			SP_RunStp50: // Do cleaning and reload from lift
				eRestartStep := SP_RunStp50;
				eRestartLoaderStep := SP_RunStp50;
				IF sRunData.sStatusLoader = RS_WaitRequest THEN
					// Check if table can be cleaned
					IF sRunData.sStatusTable = RS_WaitRequest AND NOT bTableIsClean THEN
						// Clean the table
						sRunData.eCmdTable := RCT_Clean;
					END_IF
					IF bNeedNewPart THEN			// HFO : add "or sProdLot.dProdQty < sProdLot.dLotQty" to pearl the 2 last pieces
						IF NOT sRunData.TDataLoader.aTPartData[0].bPartPresent AND NOT bTablePos2NeedPart THEN
							sRunData.TDataLoader.eModule := LMP_Lift1;
							sRunData.TDataLoader.eTaker := LH_Head1;
							sRunData.eCmdLoader := RCLo_PrepareTakePart;
							eManagerStep := SP_RunStp55;
						ELSIF NOT sRunData.TDataLoader.aTPartData[1].bPartPresent THEN
							sRunData.TDataLoader.eModule := LMP_Lift1;
							sRunData.TDataLoader.eTaker := LH_Head2;
							sRunData.eCmdLoader := RCLo_PrepareTakePart;
							eManagerStep := SP_RunStp55;
						ELSIF sRunData.sStatusTable = RS_WaitRequest THEN
							bTableIsClean := TRUE;
							eManagerStep := SP_RunStp70;
						END_IF	
					ELSIF sRunData.sStatusTable = RS_WaitRequest AND sProdLot.dProdQty < sProdLot.dLotQty THEN			// TODO : HFO, add elseif to pearl the 2 last pieces
						bTableIsClean := TRUE;
						eManagerStep := SP_RunStp70;
					ELSE
						eManagerStep := SP_RunStp80;
						// eManagerStep := SP_RunStp160; 	// purging
					END_IF
				END_IF				
			SP_RunStp55:
				IF sRunData.sStatusLoader = RS_WaitRequest THEN
					sRunData.eCmdLoader := RCLo_TakePart;
					eManagerStep := SP_RunStp60;
				END_IF
			SP_RunStp60:
				IF sRunData.sStatusLoader = RS_WaitRequest 
						AND sRunData.sStatusTable = RS_WaitRequest THEN
					bTableIsClean := TRUE;
					eManagerStep := SP_RunStp50;
				END_IF
			SP_RunStp70: (* Drop part on layering *)
				IF sRunData.sStatusTable = RS_WaitRequest THEN
					eRestartStep := SP_RunStp70;
					eRestartLoaderStep := SP_RunStp70;
					IF sRunData.TDataLoader.aTPartData[0].bPartPresent THEN
						IF sRunData.TDataLoader.aTPartData[0].bToReject THEN
							sRunData.TDataLoader.eModule := LMP_Reject;
							sRunData.TDataLoader.eTaker := LH_Head1;
							sRunData.eCmdLoader := RCLo_PrepareDropPart;
							eManagerStep := SP_RunStp150;
						ELSE
							sRunData.TDataLoader.eModule := LMP_Table;
							sRunData.TDataLoader.eTaker := LH_Head1;
							sRunData.TDataLoader.iLayringPos := 0;
							sRunData.eCmdLoader := RCLo_PrepareDropPart;
							eManagerStep := SP_RunStp75;
						END_IF
					ELSIF sRunData.TDataLoader.aTPartData[1].bPartPresent THEN
						IF sRunData.TDataLoader.aTPartData[1].bToReject THEN
							sRunData.TDataLoader.eModule := LMP_Reject;
							sRunData.TDataLoader.eTaker := LH_Head2;
							sRunData.eCmdLoader := RCLo_PrepareDropPart;
							bTablePos2NeedPart := TRUE;
							eManagerStep := SP_RunStp150;
						ELSE
							sRunData.TDataLoader.eModule := LMP_Table;
							sRunData.TDataLoader.eTaker := LH_Head2;
							sRunData.TDataLoader.iLayringPos := 1;
							sRunData.eCmdLoader := RCLo_PrepareDropPart;
							bTablePos2NeedPart := FALSE;
							eManagerStep := SP_RunStp75;
						END_IF
					ELSE
						// Loading finished, turn table
						eManagerStep := SP_RunStp80;
					END_IF
				END_IF
			SP_RunStp75:
				IF sRunData.sStatusLoader = RS_WaitRequest THEN
					sRunData.TDataTable.iGiveTakeLayeringPosition := sRunData.TDataLoader.iLayringPos;
					sRunData.eCmdLoader := RCLo_GivePart;
					sRunData.eCmdTable := RCT_TakePart;
					eManagerStep := SP_RunStp77;
				END_IF
			SP_RunStp77:
				IF sRunData.sStatusLoader = RS_WaitRequest AND  sRunData.sStatusTable = RS_WaitRequest  THEN
					eManagerStep := SP_RunStp70;
				END_IF		
			SP_RunStp80:
				IF sRunData.sStatusLoader = RS_WaitRequest AND  sRunData.sStatusTable = RS_WaitRequest  THEN
					sRunData.eCmdLoader := RCLo_MoveToSafe;
					eManagerStep := SP_RunStp85;
				END_IF		
			SP_RunStp85:
				IF sRunData.sStatusLoader = RS_WaitRequest AND bPearlingFinishOnTableSide THEN
					(* Pearling finish *)
					bReadyForPearling := FALSE;
					eManagerStep := SP_RunStp90;
				END_IF
			SP_RunStp90:
				eRestartStep := SP_RunStp96;
				eRestartLoaderStep := SP_RunStp93;
				sRunData.eCmdTable := RCT_Turn;
				eWorkingTableSide := ePearlingTableSide;
				eManagerStep := SP_RunStp93;
			SP_RunStp93: (*Turning Table *)
				IF sRunData.sStatusTable = RS_ProcessRequest2 THEN
					IF iPartOnProcess = 0 AND NOT bNeedNewPart THEN
						eManagerStep := SP_RunStp300;
					ELSE
						bReadyForPearling := TRUE;
						eManagerStep := SP_RunStp96;
					END_IF
				END_IF
			SP_RunStp96: (*Cleaning Table *)
				IF sRunData.sStatusTable = RS_WaitRequest  AND  sRunData.sStatusLoader = RS_WaitRequest  THEN
					bTableIsClean := TRUE;
					eManagerStep := SP_RunStp1;
				END_IF
			SP_RunStp100: (* Unloading part on layering *)
				IF sRunData.TDataTable.aTPartData[0,0,sRunData.TDataTable.eTableSide].bPartPresent OR sRunData.TDataTable.aTPartData[1,0,sRunData.TDataTable.eTableSide].bPartPresent THEN
					eRestartStep := SP_RunStp100;
					eRestartLoaderStep := SP_RunStp100;
					sRunData.TDataLoader.eModule := LMP_Table;
					sRunData.eCmdLoader := RCLo_PrepareTakePart;
					eManagerStep := SP_RunStp105;
				ELSE
					eManagerStep := SP_RunStp1;
				END_IF
			SP_RunStp105:
				IF sRunData.sStatusLoader = RS_WaitRequest THEN
					sRunData.eCmdLoader := RCLo_TakePart;
					sRunData.TDataTable.iGiveTakeLayeringPosition := sRunData.TDataLoader.iLayringPos;
					sRunData.TDataTable.iGiveTakeLayeringOffsetPosition := sRunData.TDataLoader.iLayringOffsetPos;
					sRunData.eCmdTable := RCT_GivePart;
					eManagerStep := SP_RunStp110;
				END_IF
			SP_RunStp110:
				IF sRunData.sStatusLoader = RS_WaitRequest AND  sRunData.sStatusTable = RS_WaitRequest  THEN
					eManagerStep := SP_RunStp1;
				END_IF
			SP_RunStp150: // Give bad part to the reject
				IF sRunData.sStatusLoader = RS_WaitRequest THEN
					sRunData.eCmdLoader := RCLo_GivePart;
					eManagerStep := SP_RunStp151;
				END_IF
			SP_RunStp151:
				IF sRunData.sStatusLoader = RS_WaitRequest THEN
					eManagerStep := SP_RunStp50;
				END_IF
			SP_RunStp160: // TODO : (HFO) // Steps for purging 
				IF sRunData.sStatusLoader = RS_WaitRequest AND  sRunData.sStatusTable = RS_WaitRequest  THEN
					sRunData.eCmdLoader := RCLo_MoveToSafe;
					//eManagerStep := SP_RunStp85;
				END_IF		
			SP_RunStp200:
				IF sRunData.sStatusLoader = RS_WaitRequest THEN
					IF sRunData.TDataLoader.aTPartData[LH_Head1].bToReject THEN
						sRunData.TDataLoader.eModule := LMP_Reject;
					ELSIF sProductionCmd.TRequestSample.Activate THEN
						sRunData.TDataLoader.eModule := LMP_Sample;
						sProductionCmd.TRequestSample.Activate := FALSE;
					ELSE
						sProductionCmd.TAutoSampling.iPeriodCnt := sProductionCmd.TAutoSampling.iPeriodCnt + 1;
						IF sProductionCmd.TAutoSampling.bEnable AND (sProductionCmd.TAutoSampling.iPeriodCnt >= (sProductionCmd.TAutoSampling.iPeriod - sProductionCmd.TAutoSampling.iBatchSize)) THEN
							sRunData.TDataLoader.eModule := LMP_Sample;
							sProductionCmd.TAutoSampling.iBatchCnt := sProductionCmd.TAutoSampling.iBatchCnt + 1;
							IF sProductionCmd.TAutoSampling.iBatchCnt >= sProductionCmd.TAutoSampling.iBatchSize THEN
								sProductionCmd.TAutoSampling.iBatchCnt := 0;
								sProductionCmd.TAutoSampling.iPeriodCnt := 0;
							END_IF
						ELSE
							sRunData.TDataLoader.eModule := LMP_Lift2;
						END_IF
					END_IF
					sRunData.eCmdLoader := RCLo_PrepareDropPart;
					eManagerStep := SP_RunStp205;
				END_IF
			SP_RunStp205:
				IF sRunData.sStatusLoader = RS_WaitRequest THEN
					sRunData.eCmdLoader := RCLo_GivePart;
					eManagerStep := SP_RunStp210;
				END_IF
			SP_RunStp210:
				IF sRunData.sStatusLoader = RS_WaitRequest THEN
					bTableIsClean := TRUE;
					eManagerStep := SP_RunStp2;
				END_IF
			SP_RunStp300: (*End of recipe *)
				bReadyForPearling := FALSE;
				sRunData.eCmdLoader := RCLo_EndOfRecipe;
				eManagerStep := SP_RunStp305;
			SP_RunStp305: (*Loader in safe and lift in unload position *)
				IF sRunData.sStatusLoader = RS_WaitRequest  AND sRunData.sStatusPearling = RS_WaitRequest AND sRunData.sStatusTable = RS_WaitRequest THEN
					eManagerStep := SP_RunStp0;
				END_IF
		END_CASE
	ELSE
		CASE eManagerStep OF
			SP_InitStp1:	(*Recovery, Drop plate if we have one*)
				sRunData.eCmdPearling := RCP_CheckSharpen;
				bReadyForPearling := FALSE;
				bTableIsClean := FALSE;
				IF sRunData.TDataLoader.bPlatePresent THEN
					sRunData.eCmdLoader := RCLo_SwitchPlate;
					eManagerStep := SP_InitStp2;
				ELSE
					eManagerStep := SP_InitStp3;
				END_IF
			SP_InitStp2: (* Switch plate done *)
				IF sRunData.sStatusLoader = RS_WaitRequest THEN
					eManagerStep := SP_InitStp3;
				END_IF
			SP_InitStp3: (* Do we need a table turn ? *)
				IF  sRunData.TDataTable.eTableSide <>  eWorkingTableSide THEN
					sRunData.eCmdTable := RCT_Turn;
					eManagerStep := SP_InitStp4;
				ELSE
					eManagerStep := SP_InitStp5;
				END_IF
			SP_InitStp4:
					IF sRunData.sStatusTable = RS_WaitRequest THEN
						eManagerStep := SP_InitStp5;
					END_IF
			SP_InitStp5:
				bReadyForPearling := TRUE;
				IF sRunData.TDataLoader.aTPartData[LH_Head1].bPartPresent THEN
					eManagerStep := eRestartLoaderStep;
				ELSE
					eManagerStep := eRestartStep;
				END_IF
	(* Running Step *)
			SP_RunStp1:
				eRestartStep := SP_RunStp1;
				eRestartLoaderStep := SP_RunStp7;
				iRunLayering := 0;
				iRunLayeringOffset := 0;
				bLastPart := FALSE;
				eManagerStep := SP_RunStp3;
			SP_RunStp2:
				bLastPart := FALSE;
				IF bLayeringWithTwoParts THEN
					IF iRunLayering=0 AND iRunLayeringOffset=0 THEN
						iRunLayering := 0;
						iRunLayeringOffset := 1;
						eManagerStep := SP_RunStp3;
					ELSIF iRunLayering=0 AND iRunLayeringOffset=1 THEN
						iRunLayering := 1;
						iRunLayeringOffset := 0;
						eManagerStep := SP_RunStp3;
					ELSIF iRunLayering=1 AND iRunLayeringOffset=0 THEN
						iRunLayering := 1;
						iRunLayeringOffset := 1;
						bLastPart := TRUE;
						eManagerStep := SP_RunStp3;
					ELSE
						eManagerStep := SP_RunStp20;
					END_IF
				ELSE
					IF iRunLayering=0 AND iRunLayeringOffset=0 THEN
						iRunLayering := 1;
						iRunLayeringOffset := 0;
						bLastPart := TRUE;
						eManagerStep := SP_RunStp3;
					ELSE
						eManagerStep := SP_RunStp20;
					END_IF
				END_IF
			SP_RunStp3:
				IF sRunData.TDataTable.aTPartData[iRunLayering,iRunLayeringOffset,sRunData.TDataTable.eTableSide].bPartPresent THEN
					bTableIsClean := FALSE;
					eManagerStep := SP_RunStp4;
				ELSE
					eManagerStep := SP_RunStp2; (* Skip *)
				END_IF
			SP_RunStp4: (* Unloading part on layering*)
				sRunData.TDataLoader.eModule := LMP_Table;
				sRunData.TDataLoader.eTaker := LH_Head1;
				sRunData.TDataLoader.iLayringPos := iRunLayering;
				sRunData.TDataLoader.iLayringOffsetPos := iRunLayeringOffset;
				sRunData.eCmdLoader := RCLo_PrepareTakePart;
				eManagerStep := SP_RunStp5;
			SP_RunStp5:
				IF sRunData.sStatusLoader = RS_WaitRequest THEN
					sRunData.eCmdLoader := RCLo_TakePart;
					sRunData.TDataTable.iGiveTakeLayeringPosition := sRunData.TDataLoader.iLayringPos;
					sRunData.TDataTable.iGiveTakeLayeringOffsetPosition := sRunData.TDataLoader.iLayringOffsetPos;
					sRunData.eCmdTable := RCT_GivePart;
					eManagerStep := SP_RunStp6;
				END_IF
			SP_RunStp6:
				IF sRunData.sStatusLoader = RS_WaitRequest AND  sRunData.sStatusTable = RS_WaitRequest  THEN
					IF bLastPart AND NOT bTableIsClean THEN
						sRunData.eCmdLoader := RCLo_MoveToSafe;
					END_IF
					eManagerStep := SP_RunStp7;
				END_IF
			SP_RunStp7:
				IF sRunData.sStatusLoader = RS_WaitRequest THEN
					IF bLastPart AND NOT bTableIsClean THEN
						sRunData.eCmdTable := RCT_Clean;
					END_IF
					IF sRunData.TDataLoader.aTPartData[LH_Head1].bToReject THEN
						sRunData.TDataLoader.eModule := LMP_Reject;
					ELSIF sProductionCmd.TRequestSample.Activate THEN
						sRunData.TDataLoader.eModule := LMP_Sample;
						sProductionCmd.TRequestSample.Activate := FALSE;
					ELSE
						sProductionCmd.TAutoSampling.iPeriodCnt := sProductionCmd.TAutoSampling.iPeriodCnt + 1;
						IF sProductionCmd.TAutoSampling.bEnable AND (sProductionCmd.TAutoSampling.iPeriodCnt >= (sProductionCmd.TAutoSampling.iPeriod - sProductionCmd.TAutoSampling.iBatchSize)) THEN
							sRunData.TDataLoader.eModule := LMP_Sample;
							sProductionCmd.TAutoSampling.iBatchCnt := sProductionCmd.TAutoSampling.iBatchCnt + 1;
							IF sProductionCmd.TAutoSampling.iBatchCnt >= sProductionCmd.TAutoSampling.iBatchSize THEN
								sProductionCmd.TAutoSampling.iBatchCnt := 0;
								sProductionCmd.TAutoSampling.iPeriodCnt := 0;
							END_IF
						ELSE
							sRunData.TDataLoader.eModule := LMP_Lift2;
						END_IF
					END_IF
					sRunData.eCmdLoader := RCLo_PrepareDropPart;
					eManagerStep := SP_RunStp9;
				END_IF
			SP_RunStp9:
				IF sRunData.sStatusLoader = RS_WaitRequest THEN
					sRunData.eCmdLoader := RCLo_GivePart;
					eManagerStep := SP_RunStp10;
				END_IF
			SP_RunStp10:
				IF sRunData.sStatusLoader = RS_WaitRequest THEN
					IF bUse103171OptimA1  THEN
						eManagerStep := SP_RunStp11;
					ELSE
						IF sRunData.sStatusTable = RS_WaitRequest THEN
							bTableIsClean := TRUE;
							eManagerStep := SP_RunStp2;
						END_IF
					END_IF
				END_IF
			SP_RunStp11: (* During cleaning, load part on head 2*)
				eRestartStep := SP_RunStp11;
				eRestartLoaderStep := SP_RunStp11;
				IF iPartOnProcess = 0 AND NOT bNeedNewPart THEN
					eManagerStep := SP_RunStp100;
				ELSE
					eManagerStep := SP_RunStp12;
				END_IF
			SP_RunStp12:
				sRunData.TDataLoader.eModule := LMP_Lift1;
				sRunData.TDataLoader.eTaker := LH_Head1;
				sRunData.eCmdLoader := RCLo_PrepareTakePart;
				eManagerStep := SP_RunStp13;
			SP_RunStp13:
				IF sRunData.sStatusLoader = RS_WaitRequest THEN
					sRunData.eCmdLoader := RCLo_TakePart;
					eManagerStep := SP_RunStp14;
				END_IF
			SP_RunStp14:
				IF sRunData.sStatusLoader = RS_WaitRequest THEN
					(* Check if table has finished or not *)
					IF sRunData.sStatusTable = RS_WaitRequest THEN
						eManagerStep := SP_RunStp2;
					ELSIF bUse103171OptimB5PreMoveXY THEN
						(* Move to safe to save time *)
						eManagerStep := SP_RunStp15;
					END_IF
				END_IF
			SP_RunStp15:
				eRestartStep := SP_RunStp15;
				eRestartLoaderStep := SP_RunStp15;
				sRunData.eCmdLoader := RCLo_MoveToSafe;
				eManagerStep := SP_RunStp16;
			SP_RunStp16:
				IF sRunData.sStatusLoader = RS_WaitRequest AND sRunData.sStatusTable = RS_WaitRequest THEN
					eManagerStep := SP_RunStp2;
				END_IF
	
			SP_RunStp20: (* Unloading finish, proceed cleaning*)
				eRestartStep := SP_RunStp20;
				eRestartLoaderStep := SP_RunStp20;
				IF iPartOnProcess = 0 AND NOT bNeedNewPart THEN
					eManagerStep := SP_RunStp100;
				ELSIF sRunData.sStatusTable = RS_WaitRequest THEN
					sRunData.eCmdLoader := RCLo_MoveToSafe;
					eManagerStep := SP_RunStp21;
				ELSE
					eManagerStep := SP_RunStp21;
				END_IF
			SP_RunStp21:
				IF sRunData.sStatusLoader = RS_WaitRequest THEN
					IF NOT bTableIsClean THEN
						sRunData.eCmdTable := RCT_Clean;
					END_IF
					IF bUse103171OptimA1 AND NOT sRunData.TDataLoader.aTPartData[LH_Head2].bPartPresent THEN
						eManagerStep := SP_RunStp200;
					ELSE
						eManagerStep := SP_RunStp22;
					END_IF
				END_IF
			SP_RunStp22: (*Cleaning Table*)
				IF sRunData.sStatusTable = RS_WaitRequest THEN
					bTableIsClean := TRUE;
					eManagerStep := SP_RunStp40;
				END_IF
			SP_RunStp40: (* Load layering *)
				eRestartStep := SP_RunStp40;
				eRestartLoaderStep := SP_RunStp44;
				iRunLayering := -1;
				iRunLayeringOffset := 1;
				eManagerStep := SP_RunStp41;
			SP_RunStp41:
				IF bLayeringWithTwoParts THEN
					IF bNeedNewPart OR iRunLayeringOffset=0 THEN
						IF iRunLayering=-1 THEN
							iRunLayering := 0;
							iRunLayeringOffset := 0;
							eManagerStep := SP_RunStp42;
						ELSIF iRunLayering=0 AND iRunLayeringOffset=0 THEN
							iRunLayering := 0;
							iRunLayeringOffset := 1;
							eManagerStep := SP_RunStp42;
						ELSIF iRunLayering=0 AND iRunLayeringOffset=1 THEN
							iRunLayering := 1;
							iRunLayeringOffset := 0;
							eManagerStep := SP_RunStp42;
						ELSIF iRunLayering=1 AND iRunLayeringOffset=0 THEN
							iRunLayering := 1;
							iRunLayeringOffset := 1;
							eManagerStep := SP_RunStp42;
						ELSE
							eManagerStep := SP_RunStp50;
						END_IF
					ELSE
						eManagerStep := SP_RunStp50;
					END_IF
				ELSE
					IF bNeedNewPart THEN
						IF iRunLayering=-1 THEN
							iRunLayering := 0;
							iRunLayeringOffset := 0;
							eManagerStep := SP_RunStp42;
						ELSIF iRunLayering=0 AND iRunLayeringOffset=0 THEN
							iRunLayering := 1;
							iRunLayeringOffset := 0;
							eManagerStep := SP_RunStp42;
						ELSE
							eManagerStep := SP_RunStp50;
						END_IF
					ELSE
						eManagerStep := SP_RunStp50;
					END_IF
				END_IF
			SP_RunStp42:
				IF NOT sRunData.TDataTable.aTPartData[iRunLayering,iRunLayeringOffset,sRunData.TDataTable.eTableSide].bPartPresent THEN
					bTableIsClean := FALSE;
					sRunData.TDataLoader.eModule := LMP_Lift1;
					sRunData.TDataLoader.eTaker := LH_Head1;
					sRunData.eCmdLoader := RCLo_PrepareTakePart;
					eManagerStep := SP_RunStp43;
				ELSE
					eManagerStep := SP_RunStp41; (* Skip *)
				END_IF
			SP_RunStp43:
				IF sRunData.sStatusLoader = RS_WaitRequest THEN
					sRunData.eCmdLoader := RCLo_TakePart;
					eManagerStep := SP_RunStp44;
				END_IF
			SP_RunStp44:
				IF sRunData.sStatusLoader = RS_WaitRequest THEN
					(* Check if a part was taken or not *)
					IF sRunData.TDataLoader.aTPartData[LH_Head1].bPartPresent THEN
						sRunData.TDataLoader.eModule := LMP_Table;
						sRunData.TDataLoader.iLayringPos := iRunLayering;
						sRunData.TDataLoader.iLayringOffsetPos := iRunLayeringOffset;
						sRunData.eCmdLoader := RCLo_PrepareDropPart;
						eManagerStep := SP_RunStp45;
					ELSE
						eManagerStep := SP_RunStp42;
					END_IF
				END_IF
			SP_RunStp45:
				IF sRunData.sStatusLoader = RS_WaitRequest THEN
					sRunData.eCmdLoader := RCLo_GivePart;
					sRunData.TDataTable.iGiveTakeLayeringPosition := sRunData.TDataLoader.iLayringPos;
					sRunData.TDataTable.iGiveTakeLayeringOffsetPosition := sRunData.TDataLoader.iLayringOffsetPos;
					sRunData.eCmdTable := RCT_TakePart;
					eManagerStep := SP_RunStp46;
				END_IF
			SP_RunStp46:
				IF sRunData.sStatusLoader = RS_WaitRequest AND  sRunData.sStatusTable = RS_WaitRequest  THEN
					(* Reject part if not correctly dropped *)
					IF sRunData.TDataLoader.aTPartData[LH_Head2].bPartPresent THEN
						eManagerStep := SP_RunStp47;
					ELSE
						eManagerStep := SP_RunStp41;
					END_IF
				END_IF
			SP_RunStp47:
				sRunData.TDataLoader.eModule := LMP_Reject;
				sRunData.eCmdLoader := RCLo_PrepareDropPart;
				eManagerStep := SP_RunStp48;
			SP_RunStp48:
				IF sRunData.sStatusLoader = RS_WaitRequest THEN
					sRunData.eCmdLoader := RCLo_GivePart;
					eManagerStep := SP_RunStp49;
				END_IF
			SP_RunStp49:
				IF sRunData.sStatusLoader = RS_WaitRequest THEN
					eManagerStep := SP_RunStp42;
				END_IF
			SP_RunStp50: (* Launch loader to safe *)
				eRestartStep := SP_RunStp50;
				eRestartLoaderStep := SP_RunStp50;
				sRunData.eCmdLoader := RCLo_MoveToSafe;
				eManagerStep := SP_RunStp51;
			SP_RunStp51:
				IF sRunData.sStatusLoader = RS_WaitRequest AND bPearlingFinishOnTableSide THEN
					(* Pearling finish *)
					bReadyForPearling := FALSE;
					eManagerStep := SP_RunStp52;
				END_IF
			SP_RunStp52:
				eRestartStep := SP_RunStp54;
				eRestartLoaderStep := SP_RunStp53;
				IF bDisableCleanAfterPearling  THEN
					sRunData.eCmdTable := RCT_Turn;
				ELSE
					sRunData.eCmdTable := RCT_TurnAndClean;
				END_IF
				eWorkingTableSide := ePearlingTableSide;
				eManagerStep := SP_RunStp53;
			SP_RunStp53: (*Turning Table *)
				IF sRunData.sStatusTable = RS_ProcessRequest2 THEN
					bReadyForPearling := TRUE;
					eManagerStep := SP_RunStp54;
				END_IF
			SP_RunStp54: (*Cleaning Table *)
				IF sRunData.sStatusTable = RS_WaitRequest  AND  sRunData.sStatusLoader = RS_WaitRequest  THEN
					bTableIsClean := TRUE;
					eManagerStep := SP_RunStp1;
				END_IF
			SP_RunStp100: (*End of recipe *)
				bReadyForPearling := FALSE;
				sRunData.eCmdLoader := RCLo_EndOfRecipe;
				eManagerStep := SP_RunStp101;
			SP_RunStp101: (*Loader in safe and lift in unload position *)
				IF sRunData.sStatusLoader = RS_WaitRequest  AND sRunData.sStatusPearling = RS_WaitRequest AND sRunData.sStatusTable = RS_WaitRequest THEN
					eManagerStep := SP_RunStp0;
				END_IF
	
			SP_RunStp200: (* During cleaning, load part on head 2*)
				eRestartStep := SP_RunStp200;
				eRestartLoaderStep := SP_RunStp200;
				IF iPartOnProcess = 0 AND NOT bNeedNewPart THEN
					eManagerStep := SP_RunStp100;
				ELSE
					eManagerStep := SP_RunStp240;
				END_IF
			SP_RunStp240: (* Load part on head 2 to save time*)
				eRestartStep := SP_RunStp240;
				eRestartLoaderStep := SP_RunStp244;
				eManagerStep := SP_RunStp241;
			SP_RunStp241:
				sRunData.TDataLoader.eModule := LMP_Lift1;
				sRunData.TDataLoader.eTaker := LH_Head2;
				sRunData.eCmdLoader := RCLo_PrepareTakePart;
				eManagerStep := SP_RunStp242;
			SP_RunStp242:
				IF sRunData.sStatusLoader = RS_WaitRequest THEN
					sRunData.eCmdLoader := RCLo_TakePart;
					eManagerStep := SP_RunStp244;
				END_IF
			SP_RunStp244:
				IF sRunData.sStatusLoader = RS_WaitRequest THEN
					(* Check if table has finished or not *)
					IF sRunData.sStatusTable = RS_WaitRequest THEN
						eManagerStep := SP_RunStp1;
					ELSIF bUse103171OptimB5PreMoveXY THEN
						(* Move to safe to save time *)
						eManagerStep := SP_RunStp245;
					END_IF
				END_IF
			SP_RunStp245:
				eRestartStep := SP_RunStp245;
				eRestartLoaderStep := SP_RunStp245;
				sRunData.eCmdLoader := RCLo_MoveToSafe;
				eManagerStep := SP_RunStp246;
			SP_RunStp246:
				IF sRunData.sStatusLoader = RS_WaitRequest AND sRunData.sStatusTable = RS_WaitRequest THEN
					eManagerStep := SP_RunStp1;
				END_IF
		END_CASE
	END_IF
	IF bLayeringWithTwoParts THEN
		IF bSimPearling AND  bReadyForPearling THEN
			IF sRunData.TDataTable.aTPartData[0,0,ePearlingTableSide].bPartPresent THEN
				sRunData.TDataTable.aTPartData[0,0,ePearlingTableSide].abPearlingDone[0,PS_SUS] := TRUE;
			END_IF
			IF sRunData.TDataTable.aTPartData[0,1,ePearlingTableSide].bPartPresent THEN
				sRunData.TDataTable.aTPartData[0,1,ePearlingTableSide].abPearlingDone[0,PS_SUS] := TRUE;
			END_IF
			IF sRunData.TDataTable.aTPartData[1,0,ePearlingTableSide].bPartPresent THEN
				sRunData.TDataTable.aTPartData[1,0,ePearlingTableSide].abPearlingDone[0,PS_SUS] := TRUE;
			END_IF
			IF sRunData.TDataTable.aTPartData[1,1,ePearlingTableSide].bPartPresent THEN
				sRunData.TDataTable.aTPartData[1,1,ePearlingTableSide].abPearlingDone[0,PS_SUS] := TRUE;
			END_IF
		ELSIF  NOT bSimPearling AND sRunData.sStatusPearling = RS_WaitRequest  AND  bReadyForPearling THEN
			IF sConfigFileData.bParallelProduction THEN
				(* Pearling does nothing, launch pearling if there is part to pearl *)
				sRunData.TDataPearling.abUseSpindle[PH_Left] := FALSE;
				sRunData.TDataPearling.abUseSpindle[PH_Right] := FALSE;
				sRunData.TDataPearling.bForceSharpenAfterPearling := FALSE;
				FOR iLayeringOffsetPos := 0 TO iMaxLayeringOffsetPos DO
					sRunData.TDataPearling.sPearlingData := sConfigFileData.asPearlingData[PS_SUS].THead[PH_Left]; (* Always same recipe when parrelle prod *)
					IF sRunData.TDataTable.aTPartData[0,iLayeringOffsetPos,ePearlingTableSide].bPartPresent AND
						sRunData.TDataPearling.abUseSpindle[PH_Left] = FALSE AND sRunData.TDataPearling.abUseSpindle[PH_Right] = FALSE AND
						NOT (sRunData.TDataTable.aTPartData[0,iLayeringOffsetPos,ePearlingTableSide].abPearlingDone[0,PS_SUS] OR sRunData.TDataTable.aTPartData[0,iLayeringOffsetPos,ePearlingTableSide].abPearlingDone[1,PS_SUS]) THEN
						sRunData.TDataPearling.abUseSpindle[PH_Left] := TRUE;
						sRunData.TDataPearling.iLayringPos := 0;
						sRunData.TDataPearling.iLayringOffsetPos := iLayeringOffsetPos;
						sRunData.TDataPearling.apsPartData[PH_Left] := ADR(sRunData.TDataTable.aTPartData[0,iLayeringOffsetPos,ePearlingTableSide]);
						IF sRunData.TDataTable.aTPartData[1,iLayeringOffsetPos,ePearlingTableSide].bPartPresent AND
							NOT (sRunData.TDataTable.aTPartData[1,iLayeringOffsetPos,ePearlingTableSide].abPearlingDone[0,PS_SUS] OR sRunData.TDataTable.aTPartData[1,iLayeringOffsetPos,ePearlingTableSide].abPearlingDone[1,PS_SUS]) THEN
								sRunData.TDataPearling.abUseSpindle[PH_Right] := TRUE;
								sRunData.TDataPearling.apsPartData[PH_Right] := ADR(sRunData.TDataTable.aTPartData[1,iLayeringOffsetPos,ePearlingTableSide]);
						END_IF
					END_IF
					IF sRunData.TDataTable.aTPartData[1,iLayeringOffsetPos,ePearlingTableSide].bPartPresent AND
						sRunData.TDataPearling.abUseSpindle[PH_Left] = FALSE AND sRunData.TDataPearling.abUseSpindle[PH_Right] = FALSE AND
						NOT (sRunData.TDataTable.aTPartData[1,iLayeringOffsetPos,ePearlingTableSide].abPearlingDone[0,PS_SUS] OR sRunData.TDataTable.aTPartData[1,iLayeringOffsetPos,ePearlingTableSide].abPearlingDone[1,PS_SUS]) THEN
							sRunData.TDataPearling.abUseSpindle[PH_Right] := TRUE;
							sRunData.TDataPearling.iLayringPos := 1;
							sRunData.TDataPearling.iLayringOffsetPos := iLayeringOffsetPos;
							sRunData.TDataPearling.apsPartData[PH_Right] := ADR(sRunData.TDataTable.aTPartData[1,iLayeringOffsetPos,ePearlingTableSide]);
					END_IF
				END_FOR
				IF sRunData.TDataPearling.abUseSpindle[PH_Left] OR sRunData.TDataPearling.abUseSpindle[PH_Right] THEN
					sRunData.eCmdPearling := RCP_Pearl;
				END_IF
			ELSE
				sRunData.TDataPearling.abUseSpindle[PH_Left] := FALSE;
				sRunData.TDataPearling.abUseSpindle[PH_Right] := FALSE;
				sRunData.TDataPearling.bForceSharpenAfterPearling := FALSE;
				FOR iLayeringPos := 0 TO 1 DO
					FOR iLayeringOffsetPos := 0 TO iMaxLayeringOffsetPos DO
						sRunData.TDataPearling.sPearlingData := sConfigFileData.asPearlingData[PS_SUS].THead[PH_Left]; (* Always same recipe when parrelle prod *)
						IF sRunData.TDataTable.aTPartData[iLayeringPos,iLayeringOffsetPos,ePearlingTableSide].bPartPresent AND
							sRunData.TDataPearling.abUseSpindle[PH_Left] = FALSE AND sRunData.TDataPearling.abUseSpindle[PH_Right] = FALSE AND
							NOT (sRunData.TDataTable.aTPartData[iLayeringPos,iLayeringOffsetPos,ePearlingTableSide].abPearlingDone[0,PS_SUS] OR sRunData.TDataTable.aTPartData[iLayeringPos,iLayeringOffsetPos,ePearlingTableSide].abPearlingDone[1,PS_SUS]) THEN
							sRunData.TDataPearling.abUseSpindle[PH_Left] := TRUE;
							sRunData.TDataPearling.iLayringPos := iLayeringPos;
							sRunData.TDataPearling.iLayringOffsetPos := iLayeringOffsetPos;
							sRunData.TDataPearling.apsPartData[PH_Left] := ADR(sRunData.TDataTable.aTPartData[iLayeringPos,iLayeringOffsetPos,ePearlingTableSide]);
						END_IF
					END_FOR
				END_FOR
				IF sRunData.TDataPearling.abUseSpindle[PH_Left] OR sRunData.TDataPearling.abUseSpindle[PH_Right] THEN
					sRunData.eCmdPearling := RCP_Pearl;
				END_IF
			END_IF
		END_IF
	ELSE
		IF bSimPearling AND  bReadyForPearling THEN
			IF sRunData.TDataTable.aTPartData[0,0,ePearlingTableSide].bPartPresent THEN
				sRunData.TDataTable.aTPartData[0,0,ePearlingTableSide].abPearlingDone[0,PS_SUS] := TRUE;
			END_IF
			IF sRunData.TDataTable.aTPartData[1,0,ePearlingTableSide].bPartPresent THEN
				sRunData.TDataTable.aTPartData[1,0,ePearlingTableSide].abPearlingDone[0,PS_SUS] := TRUE;
			END_IF
		ELSIF  NOT bSimPearling AND sRunData.sStatusPearling = RS_WaitRequest  AND  bReadyForPearling THEN
			IF sConfigFileData.bParallelProduction THEN
				(* Pearling does nothing, launch pearling if there is part to pearl *)
				sRunData.TDataPearling.abUseSpindle[PH_Left] := FALSE;
				sRunData.TDataPearling.abUseSpindle[PH_Right] := FALSE;
				sRunData.TDataPearling.bForceSharpenAfterPearling := FALSE;
				FOR iLayeringOffsetPos := 0 TO iMaxLayeringOffsetPos DO
					sRunData.TDataPearling.sPearlingData := sConfigFileData.asPearlingData[PS_SUS].THead[PH_Left]; (* Always same recipe when parrelle prod *)
					IF sRunData.TDataTable.aTPartData[0,iLayeringOffsetPos,ePearlingTableSide].bPartPresent AND
						sRunData.TDataPearling.abUseSpindle[PH_Left] = FALSE AND sRunData.TDataPearling.abUseSpindle[PH_Right] = FALSE AND
						NOT (sRunData.TDataTable.aTPartData[0,iLayeringOffsetPos,ePearlingTableSide].abPearlingDone[0,PS_SUS] OR sRunData.TDataTable.aTPartData[0,iLayeringOffsetPos,ePearlingTableSide].abPearlingDone[1,PS_SUS]) THEN
						sRunData.TDataPearling.abUseSpindle[PH_Left] := TRUE;
						sRunData.TDataPearling.iLayringPos := 0;
						sRunData.TDataPearling.iLayringOffsetPos := iLayeringOffsetPos;
						sRunData.TDataPearling.apsPartData[PH_Left] := ADR(sRunData.TDataTable.aTPartData[0,iLayeringOffsetPos,ePearlingTableSide]);
						IF sRunData.TDataTable.aTPartData[1,iLayeringOffsetPos,ePearlingTableSide].bPartPresent AND
							NOT (sRunData.TDataTable.aTPartData[1,iLayeringOffsetPos,ePearlingTableSide].abPearlingDone[0,PS_SUS] OR sRunData.TDataTable.aTPartData[1,iLayeringOffsetPos,ePearlingTableSide].abPearlingDone[1,PS_SUS]) THEN
								sRunData.TDataPearling.abUseSpindle[PH_Right] := TRUE;
								sRunData.TDataPearling.apsPartData[PH_Right] := ADR(sRunData.TDataTable.aTPartData[1,iLayeringOffsetPos,ePearlingTableSide]);
						END_IF
					END_IF
					IF sRunData.TDataTable.aTPartData[1,iLayeringOffsetPos,ePearlingTableSide].bPartPresent AND
						sRunData.TDataPearling.abUseSpindle[PH_Left] = FALSE AND sRunData.TDataPearling.abUseSpindle[PH_Right] = FALSE AND
						NOT (sRunData.TDataTable.aTPartData[1,iLayeringOffsetPos,ePearlingTableSide].abPearlingDone[0,PS_SUS] OR sRunData.TDataTable.aTPartData[1,iLayeringOffsetPos,ePearlingTableSide].abPearlingDone[1,PS_SUS]) THEN
							sRunData.TDataPearling.abUseSpindle[PH_Right] := TRUE;
							sRunData.TDataPearling.iLayringPos := 1;
							sRunData.TDataPearling.iLayringOffsetPos := iLayeringOffsetPos;
							sRunData.TDataPearling.apsPartData[PH_Right] := ADR(sRunData.TDataTable.aTPartData[1,iLayeringOffsetPos,ePearlingTableSide]);
					END_IF
				END_FOR
				IF sRunData.TDataPearling.abUseSpindle[PH_Left] OR sRunData.TDataPearling.abUseSpindle[PH_Right] THEN
					sRunData.eCmdPearling := RCP_Pearl;
				END_IF
			ELSE
				sRunData.TDataPearling.abUseSpindle[PH_Left] := FALSE;
				sRunData.TDataPearling.abUseSpindle[PH_Right] := FALSE;
				sRunData.TDataPearling.bForceSharpenAfterPearling := FALSE;
				FOR iLayeringPos := 0 TO 1 DO
					FOR iLayeringOffsetPos := 0 TO iMaxLayeringOffsetPos DO
						sRunData.TDataPearling.sPearlingData := sConfigFileData.asPearlingData[PS_SUS].THead[PH_Left]; (* Always same recipe when parrelle prod *)
						IF sRunData.TDataTable.aTPartData[iLayeringPos,iLayeringOffsetPos,ePearlingTableSide].bPartPresent AND
							sRunData.TDataPearling.abUseSpindle[PH_Left] = FALSE AND sRunData.TDataPearling.abUseSpindle[PH_Right] = FALSE AND
							NOT (sRunData.TDataTable.aTPartData[iLayeringPos,iLayeringOffsetPos,ePearlingTableSide].abPearlingDone[0,PS_SUS] OR sRunData.TDataTable.aTPartData[iLayeringPos,iLayeringOffsetPos,ePearlingTableSide].abPearlingDone[1,PS_SUS]) THEN
							sRunData.TDataPearling.abUseSpindle[PH_Left] := TRUE;
							sRunData.TDataPearling.iLayringPos := iLayeringPos;
							sRunData.TDataPearling.iLayringOffsetPos := iLayeringOffsetPos;
							sRunData.TDataPearling.apsPartData[PH_Left] := ADR(sRunData.TDataTable.aTPartData[iLayeringPos,iLayeringOffsetPos,ePearlingTableSide]);
						END_IF
					END_FOR
				END_FOR
				IF sRunData.TDataPearling.abUseSpindle[PH_Left] OR sRunData.TDataPearling.abUseSpindle[PH_Right] THEN
					sRunData.eCmdPearling := RCP_Pearl;
				END_IF
			END_IF
		END_IF
	END_IF
END_IF

iStep := eManagerStep;
bRecipeIsFinish := eManagerStep = SP_RunStp0;


(* Check config errors *)
bConfigError := (NOT bUseTurnOver AND bPearlsOnSideSous) OR (sConfigFileData.bParallelProduction AND bPearlsOnSideSous);

END_FUNCTION_BLOCK

// ---- POUs/Manager/ManagerRunTest.TcPOU
FUNCTION_BLOCK ManagerRunTest
VAR_INPUT
	sConfigFileData			: TConfigFileData;
	bFirstCycle				: BOOL;
END_VAR
VAR_OUTPUT
END_VAR
VAR_IN_OUT
	sRunData				: TRunData;
END_VAR
VAR PERSISTENT
	bTestLiftMode				: BOOL		 := FALSE;
END_VAR
VAR
	bTurnOverTurn			: BOOL;
	bTurnOverTake			: BOOL;
	bTurnOverGive			: BOOL;

	bTableTurn				: BOOL;
	bTableClean				: BOOL;
	bTableTakeHead1		: BOOL;
	bTableGiveHead1		: BOOL;
	bTableTakeHead2		: BOOL;
	bTableGiveHead2		: BOOL;


	bLoaderTakePart			: BOOL;
	bLoaderDropPart			: BOOL;
	bLoaderTakePlate		: BOOL;
	bLoaderDropPlate		: BOOL;
	bLoaderCleaningHead1	: BOOL;
	bLoaderCleaningHead2	: BOOL;
	bLoaderPrepareTakePartLift				: BOOL;
	bLoaderPrepareTakePartTableHead1		: BOOL;
	bLoaderPrepareTakePartTableHead2		: BOOL;
	bLoaderPrepareTakePartTurnOverHead2	: BOOL;

	bLoaderPrepareDropPartLiftHead1		: BOOL;
	bLoaderPrepareDropPartLiftHead2		: BOOL;
	bLoaderPrepareDropPartRejectHead1	: BOOL;
	bLoaderPrepareDropPartRejectHead2	: BOOL;
	bLoaderPrepareDropPartTurnOver		: BOOL;
	bLoaderPrepareDropPartTableHead1	: BOOL;
	bLoaderPrepareDropPartTableHead2	: BOOL;
	bLoaderMoveToSafe					: BOOL;
	bLoaderSwitchPlate					: BOOL;
	bLoaderEndOfRecipe				: BOOL;
	bLoaderScanPlateLift1Model1		: BOOL;
	bLoaderScanPlateLift2Model1		: BOOL;
	bLoaderScanPlateRejectModel1	: BOOL;
	bLoaderScanPlateLift1Model2		: BOOL;
	bLoaderScanPlateLift2Model2		: BOOL;
	bLoaderScanPlateRejectModel2	: BOOL;
	bLoaderScanPlateLift1Model3		: BOOL;

	bPearlingLayering1Head1		: BOOL;
	bPearlingLayering1Head2		: BOOL;
	bPearlingLayering2Head1		: BOOL;
	bPearlingLayering2Head2		: BOOL;
	bPearlingChangeChuck		: BOOL;
	bPearlingLayering12Head12	: BOOL;

	bLift1MoveToPlate			: BOOL;
	bLift1MoveToLoadPlate		: BOOL;
	bLift1MoveToOpenDrawer		: BOOL;

	bLift2MoveToPlate			: BOOL;
	bLift2MoveToLoadPlate		: BOOL;
	bLift2MoveToOpenDrawer		: BOOL;

	bStartStepMode		: BOOL;
	bDoStepMode		: BOOL;

	ePearlingTableSide		: TTableSide;

	eManagerStep			: TModuleSteps := SP_RunStp10;

END_VAR

sRunData.eCmdTurnOver := RCTO_None;
sRunData.eCmdTable := RCT_None;
sRunData.eCmdLoader := RCLo_None;
sRunData.eCmdPearling := RCP_None;
IF bTestLiftMode THEN
	sRunData.eCmdLift1 := RCL_None;
	sRunData.eCmdLift2 := RCL_None;
END_IF


IF sRunData.TDataTable.eTableSide = TS_A THEN
	ePearlingTableSide := TS_B;
ELSE
	ePearlingTableSide := TS_A;
END_IF

IF bFirstCycle THEN
	bDoStepMode := FALSE;
END_IF
(* For testing purpose *)
IF bTurnOverTurn THEN
	sRunData.eCmdTurnOver := RCTO_Turn;
	bTurnOverTurn := FALSE;
END_IF
IF bTurnOverTake THEN
	sRunData.eCmdTurnOver := RCTO_TakePart;
	bTurnOverTake := FALSE;
END_IF
IF bTurnOverGive THEN
	sRunData.eCmdTurnOver := RCTO_GivePart;
	bTurnOverGive := FALSE;
END_IF
IF bTableTurn THEN
	sRunData.eCmdTable := RCT_Turn;
	bTableTurn := FALSE;
END_IF
IF bTableClean THEN
	sRunData.eCmdTable := RCT_Clean;
	bTableClean := FALSE;
END_IF
IF bTableTakeHead1 THEN
	sRunData.TDataTable.iGiveTakeLayeringPosition := 0;
	sRunData.TDataTable.iGiveTakeLayeringOffsetPosition := 0;
	sRunData.eCmdTable := RCT_TakePart;
	bTableTakeHead1 := FALSE;
END_IF
IF bTableGiveHead1 THEN
	sRunData.TDataTable.iGiveTakeLayeringPosition := 0;
	sRunData.TDataTable.iGiveTakeLayeringOffsetPosition := 0;
	sRunData.eCmdTable := RCT_GivePart;
	bTableGiveHead1 := FALSE;
END_IF


IF bTableTakeHead2 THEN
	sRunData.TDataTable.iGiveTakeLayeringPosition := 1;
	sRunData.TDataTable.iGiveTakeLayeringOffsetPosition := 0;
	sRunData.eCmdTable := RCT_TakePart;
	bTableTakeHead2 := FALSE;
END_IF
IF bTableGiveHead2 THEN
	sRunData.TDataTable.iGiveTakeLayeringPosition := 1;
	sRunData.TDataTable.iGiveTakeLayeringOffsetPosition := 0;
	sRunData.eCmdTable := RCT_GivePart;
	bTableGiveHead2 := FALSE;
END_IF

IF bLoaderTakePart THEN
	sRunData.eCmdLoader := RCLo_TakePart;
	bLoaderTakePart := FALSE;
END_IF
IF bLoaderDropPart THEN
	sRunData.eCmdLoader := RCLo_GivePart;
	bLoaderDropPart := FALSE;
END_IF
IF bLoaderTakePlate THEN
	sRunData.eCmdLoader := RCLo_TakePlate;
	bLoaderTakePlate := FALSE;
END_IF
IF bLoaderDropPlate THEN
	sRunData.eCmdLoader := RCLo_GivePlate;
	bLoaderDropPlate := FALSE;
END_IF
IF bLoaderCleaningHead1 THEN
	sRunData.eCmdLoader := RCLo_Cleaning;
	sRunData.TDataLoader.eTaker := LH_Head1;
	bLoaderCleaningHead1 := FALSE;
END_IF
IF bLoaderCleaningHead2 THEN
	sRunData.eCmdLoader := RCLo_Cleaning;
	sRunData.TDataLoader.eTaker := LH_Head2;
	bLoaderCleaningHead2 := FALSE;
END_IF
IF bLoaderPrepareTakePartLift THEN
	sRunData.TDataLoader.eModule := LMP_Lift1;
	sRunData.TDataLoader.eTaker := LH_Head1;
	sRunData.eCmdLoader := RCLo_PrepareTakePart;
	bLoaderPrepareTakePartLift := FALSE;
END_IF
IF bLoaderPrepareTakePartTableHead1 THEN
	sRunData.TDataLoader.eModule := LMP_Table;
	sRunData.TDataLoader.eTaker := LH_Head1;
	sRunData.TDataLoader.iLayringPos := 0;
	sRunData.TDataLoader.iLayringOffsetPos := 0;
	sRunData.eCmdLoader := RCLo_PrepareTakePart;
	bLoaderPrepareTakePartTableHead1 := FALSE;
END_IF
IF bLoaderPrepareTakePartTableHead2 THEN
	sRunData.TDataLoader.eModule := LMP_Table;
	sRunData.TDataLoader.eTaker := LH_Head2;
	sRunData.TDataLoader.iLayringPos := 1;
	sRunData.TDataLoader.iLayringOffsetPos := 0;
	sRunData.eCmdLoader := RCLo_PrepareTakePart;
	bLoaderPrepareTakePartTableHead2 := FALSE;
END_IF
IF bLoaderPrepareTakePartTurnOverHead2 THEN
	sRunData.TDataLoader.eModule := LMP_TurnOverFix;
	sRunData.TDataLoader.eTaker := LH_Head2;
	sRunData.eCmdLoader := RCLo_PrepareTakePart;
	bLoaderPrepareTakePartTurnOverHead2 := FALSE;
END_IF
IF bLoaderPrepareDropPartLiftHead1 THEN
	sRunData.TDataLoader.eModule := LMP_Lift2;
	sRunData.TDataLoader.eTaker := LH_Head1;
	sRunData.eCmdLoader := RCLo_PrepareDropPart;
	bLoaderPrepareDropPartLiftHead1 := FALSE;
END_IF
IF bLoaderPrepareDropPartLiftHead2 THEN
	sRunData.TDataLoader.eModule := LMP_Lift2;
	sRunData.TDataLoader.eTaker := LH_Head2;
	sRunData.eCmdLoader := RCLo_PrepareDropPart;
	bLoaderPrepareDropPartLiftHead2 := FALSE;
END_IF
IF bLoaderPrepareDropPartRejectHead1 THEN
	sRunData.TDataLoader.eModule := LMP_Reject;
	sRunData.TDataLoader.eTaker := LH_Head1;
	sRunData.eCmdLoader := RCLo_PrepareDropPart;
	bLoaderPrepareDropPartRejectHead1 := FALSE;
END_IF
IF bLoaderPrepareDropPartRejectHead2 THEN
	sRunData.TDataLoader.eModule := LMP_Reject;
	sRunData.TDataLoader.eTaker := LH_Head2;
	sRunData.eCmdLoader := RCLo_PrepareDropPart;
	bLoaderPrepareDropPartRejectHead2 := FALSE;
END_IF
IF bLoaderPrepareDropPartTurnOver THEN
	sRunData.TDataLoader.eModule := LMP_TurnOverArm;
	sRunData.TDataLoader.eTaker := LH_Head1;
	sRunData.eCmdLoader := RCLo_PrepareDropPart;
	bLoaderPrepareDropPartTurnOver := FALSE;
END_IF
IF bLoaderPrepareDropPartTableHead1 THEN
	sRunData.TDataLoader.eModule := LMP_Table;
	sRunData.TDataLoader.eTaker := LH_Head1;
	sRunData.TDataLoader.iLayringPos := 0;
	sRunData.TDataLoader.iLayringOffsetPos := 0;
	sRunData.eCmdLoader := RCLo_PrepareDropPart;
	bLoaderPrepareDropPartTableHead1 := FALSE;
END_IF
IF bLoaderPrepareDropPartTableHead2 THEN
	sRunData.TDataLoader.eModule := LMP_Table;
	sRunData.TDataLoader.eTaker := LH_Head2;
	sRunData.TDataLoader.iLayringPos := 1;
	sRunData.TDataLoader.iLayringOffsetPos := 0;
	sRunData.eCmdLoader := RCLo_PrepareDropPart;
	bLoaderPrepareDropPartTableHead2 := FALSE;
END_IF
IF bLoaderMoveToSafe THEN
	sRunData.eCmdLoader := RCLo_MoveToSafe;
	bLoaderMoveToSafe := FALSE;
END_IF
IF bLoaderSwitchPlate THEN
	sRunData.eCmdLoader := RCLo_SwitchPlate;
	bLoaderSwitchPlate := FALSE;
END_IF
IF bLoaderEndOfRecipe THEN
	sRunData.eCmdLoader := RCLo_EndOfRecipe;
	bLoaderEndOfRecipe := FALSE;
END_IF
IF bLoaderScanPlateLift1Model1 THEN
	sRunData.TDataLoader.eModule := LMP_Lift1;
	sRunData.TDataLoader.iScanModel := 0;
	sRunData.eCmdLoader := RCLo_ScanPlate;
	bLoaderScanPlateLift1Model1 := FALSE;
END_IF
IF bLoaderScanPlateLift2Model1 THEN
	sRunData.TDataLoader.eModule := LMP_Lift2;
	sRunData.TDataLoader.iScanModel := 0;
	sRunData.eCmdLoader := RCLo_ScanPlate;
	bLoaderScanPlateLift2Model1 := FALSE;
END_IF
IF bLoaderScanPlateRejectModel1 THEN
	sRunData.TDataLoader.eModule := LMP_Reject;
	sRunData.TDataLoader.iScanModel := 0;
	sRunData.eCmdLoader := RCLo_ScanPlate;
	bLoaderScanPlateRejectModel1 := FALSE;
END_IF

IF bLoaderScanPlateLift1Model2 THEN
	sRunData.TDataLoader.eModule := LMP_Lift1;
	sRunData.TDataLoader.iScanModel := 1;
	sRunData.eCmdLoader := RCLo_ScanPlate;
	bLoaderScanPlateLift1Model2 := FALSE;
END_IF
IF bLoaderScanPlateLift2Model2 THEN
	sRunData.TDataLoader.eModule := LMP_Lift2;
	sRunData.TDataLoader.iScanModel := 1;
	sRunData.eCmdLoader := RCLo_ScanPlate;
	bLoaderScanPlateLift2Model2 := FALSE;
END_IF
IF bLoaderScanPlateRejectModel2 THEN
	sRunData.TDataLoader.eModule := LMP_Reject;
	sRunData.TDataLoader.iScanModel := 1;
	sRunData.eCmdLoader := RCLo_ScanPlate;
	bLoaderScanPlateRejectModel2 := FALSE;
END_IF
IF bLoaderScanPlateLift1Model3 THEN
	sRunData.TDataLoader.eModule := LMP_Lift1;
	sRunData.TDataLoader.iScanModel := 2;
	sRunData.eCmdLoader := RCLo_ScanPlate;
	bLoaderScanPlateLift1Model3 := FALSE;
END_IF


IF bPearlingLayering1Head1 THEN
	sRunData.TDataPearling.sPearlingData := sConfigFileData.asPearlingData[PS_SUS].THead[PH_Left];
	sRunData.TDataPearling.abUseSpindle[PH_Left] := TRUE;
	sRunData.TDataPearling.abUseSpindle[PH_Right] := FALSE;
	sRunData.TDataPearling.iLayringPos := 0;
	sRunData.TDataPearling.iLayringOffsetPos := 0;
	sRunData.TDataPearling.apsPartData[PH_Left] := ADR(sRunData.TDataTable.aTPartData[0,0,ePearlingTableSide]);
	sRunData.eCmdPearling := RCP_Pearl;
	bPearlingLayering1Head1 := FALSE;
END_IF

IF bPearlingLayering1Head2 THEN
	sRunData.TDataPearling.sPearlingData := sConfigFileData.asPearlingData[PS_SUS].THead[PH_Right];
	sRunData.TDataPearling.abUseSpindle[PH_Left] := FALSE;
	sRunData.TDataPearling.abUseSpindle[PH_Right] := TRUE;
	sRunData.TDataPearling.iLayringPos := 0;
	sRunData.TDataPearling.iLayringOffsetPos := 0;
	sRunData.TDataPearling.apsPartData[PH_Right] := ADR(sRunData.TDataTable.aTPartData[0,0,ePearlingTableSide]);
	sRunData.eCmdPearling := RCP_Pearl;
	bPearlingLayering1Head2 := FALSE;
END_IF

IF bPearlingLayering2Head1 THEN
	sRunData.TDataPearling.sPearlingData := sConfigFileData.asPearlingData[PS_SOUS].THead[PH_Left];
	sRunData.TDataPearling.abUseSpindle[PH_Left] := TRUE;
	sRunData.TDataPearling.abUseSpindle[PH_Right] := FALSE;
	sRunData.TDataPearling.iLayringPos := 1;
	sRunData.TDataPearling.iLayringOffsetPos := 0;
	sRunData.TDataPearling.apsPartData[PH_Left] := ADR(sRunData.TDataTable.aTPartData[1,0,ePearlingTableSide]);
	sRunData.eCmdPearling := RCP_Pearl;
	bPearlingLayering2Head1 := FALSE;
END_IF

IF bPearlingLayering2Head2 THEN
	sRunData.TDataPearling.sPearlingData := sConfigFileData.asPearlingData[PS_SOUS].THead[PH_Right];
	sRunData.TDataPearling.abUseSpindle[PH_Left] := FALSE;
	sRunData.TDataPearling.abUseSpindle[PH_Right] := TRUE;
	sRunData.TDataPearling.iLayringPos := 1;
	sRunData.TDataPearling.iLayringOffsetPos := 0;
	sRunData.TDataPearling.apsPartData[PH_Right] := ADR(sRunData.TDataTable.aTPartData[1,0,ePearlingTableSide]);
	sRunData.eCmdPearling := RCP_Pearl;
	bPearlingLayering2Head2 := FALSE;
END_IF

IF bPearlingLayering12Head12 THEN
	sRunData.TDataPearling.sPearlingData := sConfigFileData.asPearlingData[PS_SUS].THead[PH_Left];
	sRunData.TDataPearling.abUseSpindle[PH_Left] := TRUE;
	sRunData.TDataPearling.abUseSpindle[PH_Right] := TRUE;
	sRunData.TDataPearling.iLayringPos := 0;
	sRunData.TDataPearling.iLayringOffsetPos := 0;
	sRunData.TDataPearling.apsPartData[PH_Left] := ADR(sRunData.TDataTable.aTPartData[0,0,ePearlingTableSide]);
	sRunData.TDataPearling.apsPartData[PH_Right] := ADR(sRunData.TDataTable.aTPartData[1,0,ePearlingTableSide]);
	sRunData.eCmdPearling := RCP_Pearl;
	bPearlingLayering12Head12 := FALSE;
END_IF

IF bPearlingChangeChuck THEN
	sRunData.eCmdPearling := RCP_ChangeChuck;
	bPearlingChangeChuck := FALSE;
END_IF

IF bTestLiftMode THEN
	IF bLift1MoveToPlate THEN
		sRunData.eCmdLift1 := RCL_MoveToPlate;
		bLift1MoveToPlate := FALSE;
	END_IF
	IF bLift1MoveToLoadPlate THEN
		sRunData.eCmdLift1 := RCL_MoveToLoadPlate;
		bLift1MoveToLoadPlate := FALSE;
	END_IF
	IF bLift1MoveToOpenDrawer THEN
		sRunData.eCmdLift1 := RCL_MoveToOpenDrawer;
		bLift1MoveToOpenDrawer := FALSE;
	END_IF
	
	
	IF bLift2MoveToPlate THEN
		sRunData.eCmdLift2 := RCL_MoveToPlate;
		bLift2MoveToPlate := FALSE;
	END_IF
	IF bLift2MoveToLoadPlate THEN
		sRunData.eCmdLift2 := RCL_MoveToLoadPlate;
		bLift2MoveToLoadPlate := FALSE;
	END_IF
	IF bLift2MoveToOpenDrawer THEN
		sRunData.eCmdLift2 := RCL_MoveToOpenDrawer;
		bLift2MoveToOpenDrawer := FALSE;
	END_IF
END_IF
	
IF bStartStepMode THEN
	bDoStepMode := TRUE;
	eManagerStep := SP_RunStp10;
	bStartStepMode := FALSE;
END_IF

IF bDoStepMode THEN
	CASE eManagerStep OF
		SP_RunStp10: (* Unloading part on layering 0 *)
			IF sRunData.TDataTable.aTPartData[0,0,sRunData.TDataTable.eTableSide].bPartPresent THEN
				eManagerStep := SP_RunStp11;
			ELSE
				eManagerStep := SP_RunStp40;(* Skip *)
			END_IF
		SP_RunStp11:
			sRunData.TDataLoader.eModule := LMP_Table;
			sRunData.TDataLoader.eTaker := LH_Head1;
			sRunData.TDataLoader.iLayringPos := 0;
			sRunData.TDataLoader.iLayringOffsetPos := 0;
			sRunData.eCmdLoader := RCLo_PrepareTakePart;
			eManagerStep := SP_RunStp12;
		SP_RunStp12:
			IF sRunData.sStatusLoader = RS_WaitRequest THEN
				sRunData.eCmdLoader := RCLo_TakePart;
				sRunData.TDataTable.iGiveTakeLayeringPosition := sRunData.TDataLoader.iLayringPos;
				sRunData.TDataTable.iGiveTakeLayeringOffsetPosition := sRunData.TDataLoader.iLayringOffsetPos;
				sRunData.eCmdTable := RCT_GivePart;
				eManagerStep := SP_RunStp13;
			END_IF
		SP_RunStp13:
			IF sRunData.sStatusLoader = RS_WaitRequest AND  sRunData.sStatusTable = RS_WaitRequest  THEN
				sRunData.TDataLoader.eModule := LMP_Lift2;
				sRunData.eCmdLoader := RCLo_PrepareDropPart;
				eManagerStep := SP_RunStp15;
			END_IF
		SP_RunStp15:
			IF sRunData.sStatusLoader = RS_WaitRequest THEN
				sRunData.eCmdLoader := RCLo_GivePart;
				eManagerStep := SP_RunStp16;
			END_IF
		SP_RunStp16:
			IF sRunData.sStatusLoader = RS_WaitRequest THEN
				eManagerStep := SP_RunStp40;
			END_IF
		SP_RunStp40: (* Load layering 1 *)
			IF NOT sRunData.TDataTable.aTPartData[0,0,sRunData.TDataTable.eTableSide].bPartPresent THEN
				sRunData.TDataLoader.eModule := LMP_Lift1;
				sRunData.TDataLoader.eTaker := LH_Head1;
				sRunData.eCmdLoader := RCLo_PrepareTakePart;
				eManagerStep := SP_RunStp41;
			ELSE
				eManagerStep := SP_RunStp10; (* Skip *)
			END_IF
		SP_RunStp41:
			IF sRunData.sStatusLoader = RS_WaitRequest THEN
				sRunData.eCmdLoader := RCLo_TakePart;
				eManagerStep := SP_RunStp42;
			END_IF
		SP_RunStp42:
			IF sRunData.sStatusLoader = RS_WaitRequest THEN
				sRunData.TDataLoader.eModule := LMP_Table;
				sRunData.TDataLoader.iLayringPos := 0;
				sRunData.TDataLoader.iLayringOffsetPos := 0;
				sRunData.eCmdLoader := RCLo_PrepareDropPart;
				eManagerStep := SP_RunStp43;
			END_IF
		SP_RunStp43:
			IF sRunData.sStatusLoader = RS_WaitRequest THEN
				sRunData.eCmdLoader := RCLo_GivePart;
				sRunData.TDataTable.iGiveTakeLayeringPosition := sRunData.TDataLoader.iLayringPos;
				sRunData.TDataTable.iGiveTakeLayeringOffsetPosition := sRunData.TDataLoader.iLayringOffsetPos;
				sRunData.eCmdTable := RCT_TakePart;
				eManagerStep := SP_RunStp44;
			END_IF
		SP_RunStp44:
			IF sRunData.sStatusLoader = RS_WaitRequest AND  sRunData.sStatusTable = RS_WaitRequest  THEN
				eManagerStep := SP_RunStp10;
			END_IF

	END_CASE
END_IF

END_FUNCTION_BLOCK

// ---- POUs/utils/StopWatch.TcPOU
FUNCTION_BLOCK StopWatch
VAR_INPUT
	bRun		: BOOL;
	bReset 		: BOOL;
	bSet		: BOOL;
	tSetTime		: TIME;
END_VAR
VAR_OUTPUT
	TElapsed	: TIME					:= t#0s;
END_VAR
VAR
	TTimer		: TON;
	TTotal		: TIME					:= t#0s;
	bLastRun	: BOOL;
END_VAR

IF bReset THEN
	TElapsed := t#0s;
	TTotal := t#0s;
	TTimer(IN := FALSE);
	IF bRun THEN
		TTimer(IN := TRUE,PT := t#49d);
	END_IF
ELSIF bSet THEN
	TTotal := tSetTime;
	TElapsed := TTotal;
	TTimer(IN := FALSE);
	IF bRun THEN
		TTimer(IN := TRUE,PT := t#49d);
	END_IF
ELSE
	IF bRun THEN
		TTimer(IN := TRUE,PT := t#49d);
	END_IF
	IF bRun <> bLastRun THEN
		bLastRun := bRun;
		IF NOT bRun THEN
			TTotal := TTotal + TTimer.ET;
			TTimer(IN := FALSE);
		END_IF
	END_IF
	IF bRun THEN
		TElapsed := TTotal + TTimer.ET;
	ELSE
		TElapsed := TTotal;
	END_IF
END_IF

END_FUNCTION_BLOCK

// ---- POUs/utils/MTBFCounter.TcPOU
FUNCTION_BLOCK MTBFCounter
VAR_INPUT
	bStart 				: BOOL;
	bReset 				: BOOL;
END_VAR
VAR_OUTPUT
	dwSeconds			: DWORD;
END_VAR
VAR PERSISTENT
	TRunningTime		: TIME					:= t#0s;
	dwRunningHours		: DWORD				:= 0;
END_VAR
VAR
	TRunningTimer		: TON;
END_VAR

IF bReset THEN
	TRunningTime := t#0s;
	dwRunningHours := 0;
	TRunningTimer(IN := FALSE);
ELSE
	IF bStart AND NOT TRunningTimer.Q THEN
		TRunningTimer(IN := TRUE,PT := t#1m);
	ELSE
		TRunningTime := TRunningTime + TRunningTimer.ET;
		TRunningTimer(IN := FALSE);
		IF bStart THEN TRunningTimer(IN := TRUE,PT := t#6000m); END_IF
	END_IF

	IF (TRunningTime > t#60m) THEN
		dwRunningHours := dwRunningHours + 1;
		TRunningTime := TRunningTime - t#60m;
	END_IF
END_IF
dwSeconds := dwRunningHours*60*60 + TIME_TO_DWORD(TRunningTime + TRunningTimer.ET )/1000;

END_FUNCTION_BLOCK

// ---- POUs/utils/RunningCounter.TcPOU
FUNCTION_BLOCK RunningCounter
VAR_INPUT
	bStart 				: BOOL;
	bReset 				: BOOL;
END_VAR
VAR_OUTPUT
	bHoursTrig			: BOOL;
	dwHours				: DWORD;
END_VAR
VAR PERSISTENT
	TRunningTime		: TIME					:= t#0s;
	dwRunningHours		: DWORD				:= 0;
END_VAR
VAR
	TRunningTimer		: TON;
END_VAR

bHoursTrig := FALSE;
IF bReset THEN
	TRunningTime := t#0s;
	dwRunningHours := 0;
	TRunningTimer(IN := FALSE);
ELSE
	IF bStart AND NOT TRunningTimer.Q THEN
		TRunningTimer(IN := TRUE,PT := t#1m);
	ELSE
		TRunningTime := TRunningTime + TRunningTimer.ET;
		TRunningTimer(IN := FALSE);
		IF bStart THEN TRunningTimer(IN := TRUE,PT := t#6000m); END_IF
	END_IF

	IF (TRunningTime > t#60m) THEN
		dwRunningHours := dwRunningHours + 1;
		TRunningTime := TRunningTime - t#60m;
		bHoursTrig := TRUE;
	END_IF
END_IF
dwHours := dwRunningHours;

END_FUNCTION_BLOCK

// ---- POUs/Handlers/LoaderHdl.TcPOU
FUNCTION_BLOCK LoaderHdl

(*
	Description 	: Function bloc to handle loader
	Author			: DRE
	Date			: 22.09.2016
	Version			: 1.00

	Modifications :

*)
VAR_INPUT
	bEnable					: BOOL;
	bResetErrors			: BOOL;
	bPowerOn				: BOOL;
	eCommand				: TModuleCommands;
	bHomeX					: BOOL;
	bLimitPosX				: BOOL;
	bLimitNegX				: BOOL;
	bHomeY					: BOOL;
	bLimitPosY				: BOOL;
	bLimitNegY				: BOOL;
	bHomeZ1					: BOOL;
	bLimitPosZ1				: BOOL;
	bLimitNegZ1				: BOOL;
	bHomeZ2					: BOOL;
	bLimitPosZ2				: BOOL;
	bLimitNegZ2				: BOOL;
	iHead1VacuumFlow		: INT;
	iHead2VacuumFlow		: INT;
	bPlateVacuumIsOk		: BOOL;
	bPlateTakerIsUp			: BOOL;
	bPlateTakerIsDown		: BOOL;
	iPlateDistance			: INT;
	bStopReq				: BOOL;
	bPauseReq				: BOOL;
	sInGiveToTable			: TTaker;
	sInTakeFromTable		: TGiver;
	sInGiveToTurnOver		: TTaker;
	sInTakeFromOver			: TGiver;
	eRunCommand				: TRunCmdLoader;
	eTableSide				: TTableSide;
	sPartDataMMI			: TPartDataMMI;
	sPlateData				: TPlateData;
	eVisionRunStatus		: TRunStatus;
	eLift1RunStatus			: TRunStatus;
	eLift2RunStatus			: TRunStatus;
	eRejectRunStatus		: TRunStatus;
	sLift1RunData			: TRunDataLift;
	sLift2RunData			: TRunDataLift;
	sRejectRunData			: TRunDataReject;
	bNewPlateLift1			: BOOL;
	bNewPlateLift2			: BOOL;
	bNewPlateReject			: BOOL;
	bNewJob					: BOOL;
	bManInterlock			: BOOL;
	sVaccumSettingsHead		: TVaccumSettings;
	sVaccumSettingsPlate	: TVaccumSettings;
	TJobElapsed				: TIME;
	dwRejectPlateNb			: DWORD;
	bDisableVision			: BOOL;
	bSlowMode				: BOOL;
END_VAR
VAR_OUTPUT
	bModuleError			: BOOL;
	bZSensorOutOfRangeError	: BOOL;
	bHead1VacuumError		: BOOL;
	bHead2VacuumError		: BOOL;
	bJackError				: BOOL;
	bXAxisError				: BOOL;
	bYAxisError				: BOOL;
	bZ1AxisError			: BOOL;
	bZ2AxisError			: BOOL;
	bTAxisError				: BOOL;
	bPlateVacuumError		: BOOL;
	bActivateHead1Vacuum	: BOOL			:= FALSE;
	bActivateHead1Blowing	: BOOL			:= FALSE;
	bActivateHead2Vacuum	: BOOL			:= FALSE;
	bActivateHead2Blowing	: BOOL			:= FALSE;
	bActivatePlateVacuum	: BOOL			:= FALSE;
	bActivatePlateBlowing	: BOOL			:= FALSE;
	bMovePlateTakerUp		: BOOL			:= FALSE;
	bMovePlateTakerDown		: BOOL			:= FALSE;
	bAspirationBrushOn		: BOOL;
	sOutGiveToTable			: TGiver;
	sOutTakeFromTable		: TTaker;
	sOutGiveToTurnOver		: TGiver;
	sOutTakeFromTurnOver	: TTaker;
	eRunStatus				: TRunStatus;
	eVisionRunCmd			: TRunCmdVision;
	eLift1RunCmd			: TRunCmdLift;
	eLift2RunCmd			: TRunCmdLift;
	eRejectRunCmd			: TRunCmdReject;
	bVacuumInUse			: BOOL;
	bManInterlockOut		: BOOL;
	bManInterlockLiftOut	: BOOL;
END_VAR
VAR_IN_OUT
	sRunDataVision			: TRunDataVision;
	sRunData				: TRunDataLoader;
	sCurrentState			: TModuleData;
	TManualCmd				: TManLoader;
	sXAxisRef				: AXIS_REF;
	sYAxisRef				: AXIS_REF;
	sZ1AxisRef				: AXIS_REF;
	sZ2AxisRef				: AXIS_REF;
	sThetaAxisRef			: AXIS_REF;
	bLift1NeedsPlate		: BOOL;
	bLift1Lift1BadPlate		: BOOL;
	bLift2NeedsPlate		: BOOL;
	bRejectNeedsPlate		: BOOL;
	sHMIPartData			: TDataLog;
	sProdLot				: TProductionLot;
	sMachineCnt				: TprodCounter;
END_VAR
VAR CONSTANT
	iMaxScanVisionModelPart		: INT 		:= 2;
	iMaxScanVisionModelPlate	: INT 		:= 2;
	iVisionModelEmpty			: INT 		:= 0;
	iVisionModelPartBase		: INT 		:= 1;
	iVisionModelPlateBase		: INT 		:= 0;
	aiVisionModelPart			: ARRAY[0..iMaxScanVisionModelPart] OF INT 	:= [iVisionModelPartBase, iVisionModelPartBase, iVisionModelPartBase];
	aiVisionModelPlate			: ARRAY[0..iMaxScanVisionModelPlate] OF INT := [iVisionModelPlateBase, iVisionModelPlateBase, iVisionModelPlateBase];
	iManMoveAxisNone			: INT 		:= -1;
	alrSafePos					: ARRAY[0..4] OF LREAL 	:= [0, 0, -11, -11, 0];		(* Security positions *)
	alrCleaningOffset			: LREAL 	:= 36;
	alrYSafePosDuringRun		: LREAL 	:= 303;								(* Be carful with var alrUnsecuredArea, alrYSafePosDuringRun need to be set outside alrUnsecuredArea *)
	lrSafeTolerance 			: LREAL 	:= 2;								(* Tolerance for safety Z axis down *)
	lrPreSafeTolerance 			: LREAL 	:= 0.5;								(* Tolerance for safety Z axis down *)
	lrMaxXYMoveAllowed			: LREAL 	:= 2.1; 							(* Max move authorized when Z axis is down *)
	lrCalibrationPartAndHeadHeight				: LREAL := 15.5;
	lrCalibrationLayeringAndPartAndHeadHeight 	: LREAL := 21;
	lrCalibrationHeadSusPartHeadSousHeight 		: LREAL := 31;
	alrLiftCalibrationOffset	: ARRAY[0..2, LA_X..LA_Y] OF LREAL	:=
									[67.95,  114.95,		(* Reject Offset *)				
									67.95, 114.95,			(* Lift1 Offset *)
									67.95, 114.95];			(* Lift2 Offset *)
									//[67.95,  114.95 - 1.65,			// 1/2 plates + error mecanic (* There is a mecanic error on the adjustement part *)
									//67.95, 114.95 + 2.15,				(* Lift1 Offset *)
									//67.95, 114.95 + 2.15];			(* Lift2 Offset *)

END_VAR
VAR PERSISTENT
	iScanTryMax					: INT 		:= 2;
	alrRobotPos					: ARRAY[0..3, 0..LTP_END] OF LREAL;
	alrRobotOffset				: ARRAY[0..3, 0..LTP_END] OF LREAL;
	alrJogStep					: ARRAY[0..4] OF LREAL 		:= [5, 5, 5, 5];		(* Jog step for X,Y,Z,Theta *)
	lrSensorAdjust				: LREAL;											(* Correction on sensor in mm *)
	lrCleaningXSpeed			: LREAL 	:= 5;
	lrCleaningThetaSpeed		: LREAL 	:= 10;
	lrCleaningThetaAngle		: LREAL 	:= 45;
	lrSpeedWithPlate			: LREAL 	:= 50;
	TSensorZWaitStabTime		: TIME		:= T#100MS;
	TVisionWaitStabTime			: TIME		:= t#100ms;
	iRetryTake					: INT		:= 3;
	alrVacuumThreshold			: ARRAY[0..1] OF LREAL		:= [8, 8]; // [-0.65,-0.65];
	alrUnsecuredArea			: ARRAY[0..1, 0..1] OF LREAL := [150, 280, 520, 420];						(* Area where loader must not go [XminYmin,XmaxYmax], when value changed, be carful with var alrYSafePosDuringRun*)
	alrSecuredSafeZPos			: ARRAY[0..1] OF LREAL 		:= [-10, -10];				(* Z position to use for safety in secured area *)
	lrThetaOffsetMecDrop		: LREAL;						(* offset for drop part without using vision, not teached, it is hard writed *)
	lrXOffsetMecDrop			: LREAL;						(* offset for drop part without using vision, not teached, it is hard writed, compensate mec offset *)
	lrYOffsetMecDrop			: LREAL;
	lrZSensorCalibrationOffset	: LREAL 	:= 0;				(* Offset between Position A and the 0 plate on reject, hard coded here*)
	bUnsecuredAeraEntry 		: BOOL 		:= FALSE;

END_VAR
VAR
	alrMaxRobotSpeed		: ARRAY[0..4] OF LREAL;
	iAxis					: INT;
	iHead					: INT;
	iTeachedAxis			: INT;
	iManMoveAxis			: INT;
	alrTargetPos			: ARRAY[0..4] OF LREAL;
	eRobotXYTStatus			: TAxisState;
	aeMoveRobotCommand		: ARRAY[0..4] OF TAxisCommands	:= [5(AC_None)];
	aTRobotAxis				: ARRAY[0..4] OF StdAxis;
	TCheckJack				: FB_CheckJack1_2;
	abEnableHeadVacuum		: ARRAY[0..1] OF BOOL;
	abBypassVacuumError		: ARRAY[0..1] OF BOOL;
	abResetVacuum			: ARRAY[0..1] OF BOOL;
	aTHeadVacuum			: ARRAY[0..1] OF FB_VacuumAnalogCheck;
	bEnablePlateVacuum		: BOOL;
	TPlateVacuum			: FB_Vacuum;
	alrRobotSpeed			: ARRAY[0..4] OF LREAL;			(* X,Y,Z1,Z2,Theta *)
	alrRobotAcceleration 	: ARRAY[0..4] OF LREAL;
	alrRobotDeceleration 	: ARRAY[0..4] OF LREAL;
	alrRobotJerk 			: ARRAY[0..4] OF LREAL;
	iRobotPosition			: INT;
	iRobotOffset			: INT;
	iTeachedModeDebug		: INT; (* 0 - None, 1 Offset and Pos, 2 - Pos, 3 - Offset *)
(*	abConflictDetected		: ARRAY[0..4] OF BOOL;*)						(* DEBUG : Used to log which conflict has been detected *)
	TSensorMeasure			: ConverterLinearLimit;
	bConflictDetected		: BOOL;
	bManualZIsSafe			: BOOL;
	ZPositionTakeGive		: LREAL;
	ZPosition				: LREAL;
	bUseGiveTake			: BOOL;
	bCleaningThetaCw		: BOOL;
	bCleaningStopTheta		: BOOL;
	bCleaningFromNegToPos	: BOOL;
(*	bPrepareForDrop			: BOOL;
	lrStartX				: LREAL;
	lrStartY				: LREAL;
	lrStartTheta			: LREAL;*)
	aTPartOnPlate			: ARRAY[0..2, 0..C_MAX_NB_OF_PARTS_ON_PLATE] OF TRunDataPlate;
	iPlatePos				: INT;
	i,j						: INT;
	abResetPlateState		: ARRAY[0..2] OF BOOL := [TRUE, TRUE, TRUE];
	abCopySwitchFromPlate 	: BOOL := FALSE;
	abCopySwitchToPlate 	: BOOL := FALSE;
	bFoundPlatePos			: BOOL;
	bInvalidPlate			: BOOL;
	bPlateEmpty				: BOOL;
	eReturnStep				: TModuleSteps;
	eReturnStepSwitchPlate	: TModuleSteps;
	eReturnStepMeasureZLift	: TModuleSteps;
	eReturnStep4SecureMove	: TModuleSteps;
	iZSensorPositionScan	: INT;
	lrZSensorPosition		: ARRAY[0..1] OF LREAL;
	TSensorZWaitStab		: TON;
	bDoNothing				: BOOL;
	TVisionWaitStab			: TON;
	sInGiveToModule			: TTaker;
	sInTakeFromModule		: TGiver;
	sOutGiveToModule		: TGiver;
	sOutTakeFromModule		: TTaker;
	eScanPos				: TLoaderTeachPos;
	ePos					: TLoaderTeachPos;
	aTScanResult			: ARRAY[0..C_MAX_NB_OF_PARTS_ON_PLATE] OF TVisionPartData;
	iRetryTakeCount			: INT;
	iVisionScanModel		: INT;
	bDoPlateScan			: BOOL;
	bTakeMoveUp				: BOOL;
	bIncProdCounter			: BOOL := FALSE;
	TComputeVisionPos		: ComputeVisionPos;
	TOffsetPos				: TPositionXYTheta;
	eDropMode				: TLoaderDropMode;
	eTakeMode				: TLoaderTakeMode;
	bRetriedCompleteLiftTake	: BOOL;
	bRetryVision			: BOOL;
	alrZLiftPos				: ARRAY[0..2] OF LREAL	:= [0, 0, 0];
	lrPartX					: LREAL;
	lrPartY					: LREAL;
	iStep					: INT;
	testLD					: TLoaderModulePos;
	alrSecuredTarget		: ARRAY[0..1] OF LREAL;					// Secured XY position to reach
	iSecuredIndexFirst		: INT;									// Index of secured position to go first
	iSecuredIndexSecond		: INT;									// Index of secured position to go second
	iEntrySecuredArea 		: INT;									// Index by where we enter de secured aera
	iScanTry				: INT;
	toto 		: BOOL;
	ntiti 		: INT;
	ntata 		: INT;
	aTPartOnSwitchPlate		: ARRAY[0..C_MAX_NB_OF_PARTS_ON_PLATE] OF TRunDataPlate;
	bBadPartDetected 		:BOOL 		:= FALSE;
END_VAR

TSensorMeasure(
	iInput := iPlateDistance,
	iHardwareMin := 12710, (*V*)
	iHardwareMax := 27827, 	(*V*)
	lrSoftwareMin := -8.5,  		(*mm*)
	lrSoftwareMax := 6.5, 		(*mm*)
	lrOffset := lrSensorAdjust	(*mm*)
	);

alrRobotOffset[LTA_X,LTO_Plate] := 145;
alrRobotOffset[LTA_Y,LTO_Plate] := -42.8;

IF (NOT sCurrentState.bStepMode) THEN
	sCurrentState.bWaitStep := FALSE;
END_IF

FOR iAxis := 0 TO 4 DO
	alrMaxRobotSpeed[iAxis] := aTRobotAxis[iAxis].lrRunningSpeed;
END_FOR

// HFO : Dynamics of axis X and Y, 2 modes for acceleration, slow and max
IF NOT bSlowMode THEN // Max mode: with 0, it use default settings
	FOR i := 0 TO 1 DO 
		alrRobotAcceleration[i] := 0;
		alrRobotDeceleration[i] := 0;
		alrRobotJerk[i] := 0;
	END_FOR
ELSE // Slow mode, Change here to set the slow mode
	FOR i := 0 TO 1 DO
		alrRobotAcceleration[i] := 10000;
		alrRobotDeceleration[i] := alrRobotAcceleration[i];		// Deceleration same as acceleration
		alrRobotJerk[i] := 100000;
	END_FOR	
END_IF

(* Vision offset are always 0 if vision disabled *)
IF bDisableVision THEN
	sRunDataVision.TVisionPartData.lrX := 0;
	sRunDataVision.TVisionPartData.lrY := 0;
	//sRunDataVision.TVisionPartData.lrTheta := 0;
	sRunDataVision.TVisionPartData.lrTheta := -90;
END_IF

eVisionRunCmd := RCV_None;
eLift1RunCmd := RCL_None;
eLift2RunCmd := RCL_None;
eRejectRunCmd := RCR_None;

CASE sRunData.eModule OF
	LMP_Table:
		sInGiveToModule := sInGiveToTable;
		sInTakeFromModule := sInTakeFromTable;
	LMP_TurnOverFix,LMP_TurnOverArm:
		sInGiveToModule := sInGiveToTurnOver;
		sInTakeFromModule := sInTakeFromOver;
END_CASE

CASE eCommand OF
	MC_NoCmd :
		CASE sCurrentState.eStatus OF
			MS_Init :
				IF sCurrentState.bInError THEN
					sCurrentState.eStatus := MS_Stopped;
				ELSE
					CASE sCurrentState.eStep OF
						SP_InitStp1 :
							(* Use maximal speed *)
							alrRobotSpeed := alrMaxRobotSpeed;
							(* Check where there is parts *)
							abBypassVacuumError[0] := FALSE;
							abBypassVacuumError[1] := FALSE;
							sRunData.aTPartData[LH_Head1].bPartPresent := abEnableHeadVacuum[0];
							sRunData.aTPartData[LH_Head2].bPartPresent := abEnableHeadVacuum[1];
							sRunData.bPlatePresent := bEnablePlateVacuum;
							alrRobotSpeed := alrMaxRobotSpeed;
							IF bEnablePlateVacuum THEN
								alrRobotSpeed[LA_X] := lrSpeedWithPlate;
								alrRobotSpeed[LA_Y] := lrSpeedWithPlate;
							END_IF
							bMovePlateTakerDown := FALSE;
							bAspirationBrushOn := FALSE;
							bRetriedCompleteLiftTake := FALSE;
							sCurrentState.eStep := SP_InitStp2;
						SP_InitStp2 :
							IF bPlateTakerIsUp AND aTHeadVacuum[0].bVacuumCorrect AND aTHeadVacuum[1].bVacuumCorrect AND TPlateVacuum.bVacuumCorrect THEN
								IF bIncProdCounter THEN
									bIncProdCounter := FALSE;
									IF sRunData.aTPartData[LH_Head1].bPartPresent THEN
										sProdLot.dLoadedQty := sProdLot.dLoadedQty + 1;
									END_IF
								END_IF
								IF sCurrentState.bInitDone THEN
									sCurrentState.eStep := SP_InitStp50;
								ELSE
									//sCurrentState.eStep := SP_InitStp3;
									sCurrentState.eStep := SP_InitStp4;
								END_IF
							END_IF
						SP_InitStp3 :
(*							aeMoveRobotCommand[LA_Z1] := AC_Init;
							aeMoveRobotCommand[LA_Z2] := AC_Init;
							IF aTRobotAxis[LA_Z1].eCurrentState = AS_InPosition AND aTRobotAxis[LA_Z2].eCurrentState = AS_InPosition THEN
								sCurrentState.eStep := SP_InitStp4;
							END_IF*)
								aeMoveRobotCommand[LA_Z1] := AC_Init;
								aeMoveRobotCommand[LA_Z2] := AC_Init;
								sCurrentState.eStep := SP_InitStp4;
						SP_InitStp4 : 
(*							IF aTRobotAxis[LA_Z1].eCurrentState=AS_InPosition AND
								aTRobotAxis[LA_Z2].eCurrentState=AS_InPosition THEN
								(* Move Z to Safe *)
								alrTargetPos[LA_Z1] := alrSafePos[LA_Z1];
								alrTargetPos[LA_Z2] := alrSafePos[LA_Z2];
								aeMoveRobotCommand[LA_Z1] := AC_MoveAtAbsPos;
								aeMoveRobotCommand[LA_Z2] := AC_MoveAtAbsPos;
*)							(* Move Z Up *)
							aeMoveRobotCommand[LA_Z1] := AC_MoveLimitNeg;
							aeMoveRobotCommand[LA_Z2] := AC_MoveLimitNeg;
							sCurrentState.eStep := SP_InitStp5;
//							END_IF
						SP_InitStp5 :
(*							IF aTRobotAxis[LA_Z1].eCurrentState=AS_InPosition AND
								aTRobotAxis[LA_Z2].eCurrentState=AS_InPosition THEN
*)							IF aTRobotAxis[LA_Z1].eCurrentState=AS_OnLimitNeg AND
								aTRobotAxis[LA_Z2].eCurrentState=AS_OnLimitNeg THEN
								(* Init X / Y / Theta*)
								aeMoveRobotCommand[LA_X] := AC_Init;
								aeMoveRobotCommand[LA_Y] := AC_Init;
								aeMoveRobotCommand[LA_THETA] := AC_Init;
								sCurrentState.eStep := SP_InitStp6;
							END_IF
						SP_InitStp6:
							IF aTRobotAxis[LA_X].eCurrentState =  AS_InPosition AND aTRobotAxis[LA_Y].eCurrentState =  AS_InPosition THEN
								(* Move X/ Y to Safe *)
								alrTargetPos[LA_X] := alrSafePos[LA_X];
								alrTargetPos[LA_Y] := alrSafePos[LA_Y];
								aeMoveRobotCommand[LA_X] := AC_MoveAtAbsPos;
								aeMoveRobotCommand[LA_Y] := AC_MoveAtAbsPos;
								sCurrentState.eStep := SP_InitStp7;
							END_IF
						SP_InitStp7 :
							IF aTRobotAxis[LA_X].eCurrentState =  AS_InPosition AND aTRobotAxis[LA_Y].eCurrentState =  AS_InPosition THEN
								(* Init Z *)
								aeMoveRobotCommand[LA_Z1] := AC_Init;
								aeMoveRobotCommand[LA_Z2] := AC_Init;
								sCurrentState.eStep := SP_InitStp8;
							END_IF
						SP_InitStp8 :
							IF aTRobotAxis[LA_Z1].eCurrentState=AS_InPosition AND
								aTRobotAxis[LA_Z2].eCurrentState=AS_InPosition THEN
								(* Move Z to Safe *)
								alrTargetPos[LA_Z1] := alrSafePos[LA_Z1];
								alrTargetPos[LA_Z2] := alrSafePos[LA_Z2];
								aeMoveRobotCommand[LA_Z1] := AC_MoveAtAbsPos;
								aeMoveRobotCommand[LA_Z2] := AC_MoveAtAbsPos;
								sCurrentState.eStep := SP_InitStp9;
							END_IF
						SP_InitStp9:
							(* Wait until we are up *)
							IF (aTRobotAxis[LA_Z1].eCurrentState = AS_InPosition) AND
								(aTRobotAxis[LA_Z2].eCurrentState = AS_InPosition) THEN
								sCurrentState.eStep := SP_InitStp10;
							END_IF
						SP_InitStp10 :
							IF (aTRobotAxis[LA_THETA].eCurrentState = AS_InPosition)  THEN
								sCurrentState.eStep := SP_InitStp99;
							END_IF
						SP_InitStp50 :
							(* Move Z to Safe *)
							alrTargetPos[LA_Z1] := alrSafePos[LA_Z1];
							alrTargetPos[LA_Z2] := alrSafePos[LA_Z2];
							aeMoveRobotCommand[LA_Z1] := AC_MoveAtAbsPos;
							aeMoveRobotCommand[LA_Z2] := AC_MoveAtAbsPos;
							sCurrentState.eStep := SP_InitStp51;
						SP_InitStp51:
							(* Wait until we are up *)
							IF (aTRobotAxis[LA_Z1].eCurrentState = AS_InPosition) AND
								(aTRobotAxis[LA_Z2].eCurrentState = AS_InPosition) THEN
								(* Move X/ Y to Safe *)
								alrTargetPos[LA_X] := alrSafePos[LA_X];
								alrTargetPos[LA_Y] := alrSafePos[LA_Y];
								aeMoveRobotCommand[LA_X] := AC_MoveAtAbsPos;
								aeMoveRobotCommand[LA_Y] := AC_MoveAtAbsPos;
								sCurrentState.eStep := SP_InitStp52;
							END_IF
						SP_InitStp52:
							IF aTRobotAxis[LA_X].eCurrentState =  AS_InPosition AND aTRobotAxis[LA_Y].eCurrentState =  AS_InPosition THEN
								sCurrentState.eStep := SP_InitStp99;
							END_IF
						SP_InitStp99 :
							sCurrentState.bInitDone := TRUE;
							sCurrentState.eStep := SP_RunStp1;
							sCurrentState.eStatus := MS_Ready;
					END_CASE
				END_IF
			MS_Running :
					// Force running safe pos
					IF (NOT sCurrentState.bWaitStep)  THEN
					IF sRunData.eTaker = LH_Head1 THEN
						iHead := 0;
					ELSE
						iHead := 1;
					END_IF
					CASE sCurrentState.eStep OF
						SP_RunStp1:
							eRunStatus := RS_WaitRequest;
							CASE eRunCommand OF
								RCLo_None:
									IF bStopReq  THEN
										sCurrentState.eStatus := MS_Ready;
									ELSIF bPauseReq THEN
										sCurrentState.eStatus := MS_Paused;
									END_IF
								RCLo_TakePart:
									sCurrentState.bWaitStep := TRUE;
									sOutTakeFromModule.bReadyToTake := FALSE;
									sOutTakeFromModule.bHasTaken := FALSE;
									sCurrentState.eStep := SP_RunStp10;
								RCLo_GivePart:
									sCurrentState.bWaitStep := TRUE;
									sOutGiveToModule.bHasGiven := FALSE;
									sOutGiveToModule.bPartDataReady := FALSE;
									sCurrentState.eStep := SP_RunStp20;
								RCLo_TakePlate:
									eReturnStep := SP_RunStp1;
									sCurrentState.eStep := SP_RunStp30;
								RCLo_GivePlate:
									eReturnStep := SP_RunStp1;
									sCurrentState.eStep := SP_RunStp40;
								RCLo_MoveToSafe:
									sCurrentState.eStep := SP_RunStp50;
								RCLo_Cleaning:
									sCurrentState.eStep := SP_RunStp60;
								RCLo_SwitchPlate:
									eReturnStep := SP_RunStp1;
									sCurrentState.eStep := SP_RunStp70;
								RCLo_PrepareTakePart:
									sCurrentState.eStep := SP_RunStp100;
								RCLo_PrepareDropPart:
									sCurrentState.eStep := SP_RunStp200;
								RCLo_EndOfRecipe:
									sCurrentState.eStep := SP_RunStp400;
								RCLo_ScanPlate:
									sCurrentState.eStep := SP_RunStp410;
							END_CASE
							IF sCurrentState.eStep<> SP_RunStp1 THEN eRunStatus := RS_ProcessRequest1; END_IF
						SP_RunStp10 :  (*Take Part*)
							CASE sRunData.eModule OF
								LMP_Lift1:
									ZPosition := ZPositionTakeGive + sPartDataMMI.lrPartOffsetZLiftTake;
									bUseGiveTake := FALSE;
									eTakeMode := sPartDataMMI.eTakeModeLift;
									abBypassVacuumError[iHead] := (sPartDataMMI.lrPartOffsetZLiftBadTake > 0);
								LMP_Table,LMP_TurnOverFix:
									ZPosition := ZPositionTakeGive + sPartDataMMI.lrPartOffsetZLayeringTake;
									bUseGiveTake := TRUE;
									eTakeMode := LTM_GoDownAndVacuum;
									abBypassVacuumError[iHead] := FALSE;
								ELSE
									ZPosition := alrSecuredSafeZPos[iHead];
									bUseGiveTake := FALSE;
									eTakeMode := LTM_GoDownAndVacuum;
									abBypassVacuumError[iHead] := FALSE;
							END_CASE
							iRetryTakeCount := 1;
							bTakeMoveUp := FALSE;
							sCurrentState.eStep := SP_RunStp11;
						SP_RunStp11 :
							IF bUseGiveTake THEN
								IF sInTakeFromModule.bPartDataReady THEN
									sRunData.aTPartData[iHead] := sInTakeFromModule.TPartData;
									sRunData.aTPartData[iHead].bPartPresent := FALSE;
									sCurrentState.eStep := SP_RunStp12;
								END_IF
							ELSE
								sRunData.aTPartData[iHead] := InitNewPartData();
								sRunData.aTPartData[iHead].dwProductionInTime := TIME_TO_DWORD(TJobElapsed);
								sRunData.aTPartData[iHead].iPlateInPos := iPlatePos;
								sRunData.aTPartData[iHead].bPartPresent := FALSE;
								bIncProdCounter := TRUE;
								sCurrentState.eStep := SP_RunStp12;
							END_IF
						SP_RunStp12 :
							alrTargetPos[LA_Z1+iHead] := ZPosition;
							aeMoveRobotCommand[LA_Z1+iHead] := AC_MoveAtAbsPos;
							sCurrentState.eStep := SP_RunStp13;
						SP_RunStp13 :  (*Movement done*)
							IF aTRobotAxis[LA_Z1+iHead].lrRemainingTimeToGo < 1 AND aTRobotAxis[LA_Z1+iHead].lrRemainingTimeToGo <> 0 AND eTakeMode = LTM_VacuumAndGoDown THEN
								abEnableHeadVacuum[iHead] := TRUE;
							END_IF
							IF aTRobotAxis[LA_Z1+iHead].eCurrentState = AS_InPosition THEN
								abEnableHeadVacuum[iHead] := TRUE;
								sOutTakeFromModule.bReadyToTake := TRUE;
								sCurrentState.eStep := SP_RunStp14;
							END_IF
						SP_RunStp14 :
							(* Wait until module has given *)
							IF sInTakeFromModule.bHasGiven OR NOT bUseGiveTake THEN
								sCurrentState.eStep := SP_RunStp15;
							END_IF
						SP_RunStp15 :
							(* Check if the part is on head *)
							IF aTRobotAxis[LA_Z1+iHead].eCurrentState = AS_InPosition THEN
								IF aTHeadVacuum[iHead].bVacuumCorrect THEN
									bRetriedCompleteLiftTake := FALSE;
									abBypassVacuumError[iHead] := FALSE;
									alrTargetPos[LA_Z1+iHead] := alrSecuredSafeZPos[iHead];
									aeMoveRobotCommand[LA_Z1+iHead] := AC_MoveAtAbsPos;
									sCurrentState.eStep := SP_RunStp16;
								ELSIF aTHeadVacuum[iHead].bVacuumError AND sPartDataMMI.lrPartOffsetZLiftBadTake > 0 AND sRunData.eModule = LMP_Lift1 THEN
									IF NOT bTakeMoveUp THEN
										bTakeMoveUp := TRUE;
										abResetVacuum[iHead] := TRUE;
										abBypassVacuumError[iHead] := FALSE;
										alrTargetPos[LA_Z1+iHead] := ZPositionTakeGive - sPartDataMMI.lrPartOffsetZLiftBadTake;
										aeMoveRobotCommand[LA_Z1+iHead] := AC_MoveAtAbsPos;
									ELSIF NOT bRetriedCompleteLiftTake THEN
										(* Ask manager to retry take *)
										bRetriedCompleteLiftTake := TRUE;
										alrTargetPos[LA_Z1+iHead] := alrSecuredSafeZPos[iHead];
										aeMoveRobotCommand[LA_Z1+iHead] := AC_MoveAtAbsPos;
										sCurrentState.eStep := SP_RunStp18;
									END_IF
								END_IF
							END_IF
						SP_RunStp16 :  (*Movement done*)
							IF aTRobotAxis[LA_Z1+iHead].eCurrentState = AS_InPosition OR
									(bUse103171OptimB5MoveOnPreSafeZ AND  (aTRobotAxis[LA_Z1].lrCurrentPos < (alrSecuredSafeZPos[0]+lrPreSafeTolerance)))THEN
								IF aTHeadVacuum[iHead].bVacuumCorrect THEN
									(* Part correctly taken *)
									IF bUseGiveTake THEN
										sOutTakeFromModule.bHasTaken := TRUE;
									ELSE
										sRunData.aTPartData[iHead].dwProductionInTime := TIME_TO_DWORD(TJobElapsed);
										sRunData.aTPartData[iHead].iPlateInPos := iPlatePos;
										sProdLot.dLoadedQty := sProdLot.dLoadedQty + 1;
										bIncProdCounter := FALSE;
										IF sRunData.eModule = LMP_Lift1 THEN
											aTPartOnPlate[ LPP_Lift1,iPlatePos].ePartStatus := PPS_Absent;
										END_IF
									END_IF
									sRunData.aTPartData[iHead].bPartPresent := TRUE;
									(*IF bBadPartDetected THEN
										sRunData.aTPartData[iHead].bToReject := TRUE;
									END_IF*)
									sRunData.aTPartData[iHead].bToReject := bBadPartDetected;
									sCurrentState.eStep := SP_RunStp1;
								ELSE
									(* Part has been not taken, retry *)
									bTakeMoveUp := FALSE;
									CASE sRunData.eModule OF
										LMP_Table,LMP_TurnOverFix:
											IF iRetryTakeCount < iRetryTake THEN
												abEnableHeadVacuum[iHead] := FALSE;
												iRetryTakeCount := iRetryTakeCount + 1;
												sCurrentState.eStep := SP_RunStp17;
											END_IF
									END_CASE
								END_IF
							END_IF
						SP_RunStp17 :  (*Retry*)
							IF aTHeadVacuum[iHead].bVacuumCorrect THEN
								sCurrentState.eStep := SP_RunStp12;
							END_IF
						SP_RunStp18 :  (*Movement done*)
							IF aTRobotAxis[LA_Z1+iHead].eCurrentState = AS_InPosition THEN
								sCurrentState.eStep := SP_RunStp1;
							END_IF
						SP_RunStp20 : (*Give Part*)
							CASE sRunData.eModule OF
								LMP_Reject, LMP_Sample:
									IF sPartDataMMI.bDropInBox THEN
										ZPosition := alrRobotPos[LTA_Z,LTP_RejectBulkBox];
									ELSE
										ZPosition := ZPositionTakeGive + sPartDataMMI.lrPartOffsetZLiftDrop;
									END_IF
									IF ZPosition > aTRobotAxis[LA_Z1+iHead].lrMaxPos THEN
										ZPosition := aTRobotAxis[LA_Z1+iHead].lrMaxPos;
									END_IF
									bUseGiveTake := FALSE;
									eDropMode := LDM_DropAndGoUp;
								LMP_Lift2:
									IF sPartDataMMI.bDropInBox THEN
										ZPosition := alrRobotPos[LTA_Z,LTP_BulkBox];
									ELSE
										ZPosition := ZPositionTakeGive + sPartDataMMI.lrPartOffsetZLiftDrop;
									END_IF
									bUseGiveTake := FALSE;
									eDropMode := LDM_DropAndGoUp;
								LMP_Table:
									ZPosition := ZPositionTakeGive + sPartDataMMI.lrPartOffsetZLayeringDrop;
									bUseGiveTake := TRUE;
									eDropMode := sPartDataMMI.eDropModeTable;
								LMP_TurnOverArm:
									ZPosition := ZPositionTakeGive + sPartDataMMI.lrPartOffsetZLayeringDrop;
									bUseGiveTake := TRUE;
									eDropMode := sPartDataMMI.eDropModeTurnOver;
								ELSE
									ZPosition := alrSecuredSafeZPos[iHead];
									bUseGiveTake := FALSE;
									eDropMode := LDM_DropAndGoUp;
							END_CASE
							IF  bUseGiveTake THEN
								sOutGiveToModule.TPartData := sRunData.aTPartData[iHead];
								IF eDropMode <> LDM_WaitDownAndDrop THEN
									sOutGiveToModule.bPartDataReady := TRUE;
								END_IF
							END_IF
							sCurrentState.eStep := SP_RunStp21;
						SP_RunStp21 :
							IF sInGiveToModule.bReadyToTake  OR NOT bUseGiveTake  THEN
								alrTargetPos[LA_Z1+iHead] := ZPosition;
								aeMoveRobotCommand[LA_Z1+iHead] := AC_MoveAtAbsPos;
								sCurrentState.eStep := SP_RunStp22;
							END_IF
						SP_RunStp22 :  (*Movement done*)
							IF (sRunData.eModule = LMP_Reject OR  sRunData.eModule = LMP_Sample) AND sRejectRunData.eRejectStatus<>RS_Locked THEN
								aeMoveRobotCommand[LA_Z1+iHead] := AC_ForceStop;
							END_IF
							IF aTRobotAxis[LA_Z1+iHead].eCurrentState = AS_InPosition THEN
								sOutGiveToModule.bPartDataReady := TRUE;
								CASE eDropMode OF
									LDM_DropAndGoUp, LDM_DropAndWaitDown :
										abEnableHeadVacuum[iHead] := FALSE;
								END_CASE
								sCurrentState.eStep := SP_RunStp23;
							END_IF
						SP_RunStp23:
							(* Check if laying vacuum is disabled *)
							IF (sRunData.eModule = LMP_Reject OR  sRunData.eModule = LMP_Sample) AND sRejectRunData.eRejectStatus<>RS_Locked THEN
								aeMoveRobotCommand[LA_Z1+iHead] := AC_ForceStop;
							END_IF
							IF aTHeadVacuum[iHead].bVacuumCorrect THEN
								IF sRunData.eModule = LMP_Lift2  OR sRunData.eModule = LMP_Sample OR sRunData.eModule = LMP_Reject THEN
									sRunData.aTPartData[iHead].iPlateOutPos := iPlatePos;
									sRunData.aTPartData[iHead].dwPlateOutQRCode := dwRejectPlateNb;
									sRunData.aTPartData[iHead].dwProductionOutTime := TIME_TO_DWORD(TJobElapsed);
									sRunData.aTPartData[iHead].dwProductionTime := sRunData.aTPartData[iHead].dwProductionOutTime - sRunData.aTPartData[iHead].dwProductionInTime;
									sRunData.aTPartData[iHead].bSample := (sRunData.eModule = LMP_Sample);
									sMachineCnt.dTotal := sMachineCnt.dTotal + 1;
									sProdLot.dProdQty := sProdLot.dProdQty + 1;
									IF sRunData.eModule = LMP_Lift2 OR sRunData.eModule = LMP_Sample THEN
										sMachineCnt.dGood := sMachineCnt.dGood + 1;
										sProdLot.dGoodQty := sProdLot.dGoodQty + 1;
									END_IF
									IF sRunData.eModule = LMP_Lift2 AND NOT sPartDataMMI.bDropInBox THEN
 										aTPartOnPlate[ LPP_Lift2,iPlatePos].ePartStatus := PPS_Present;
									ELSIF sRunData.eModule = LMP_Sample THEN
										aTPartOnPlate[ LPP_Reject,iPlatePos].ePartStatus := PPS_Present;
									ELSIF sRunData.eModule = LMP_Reject THEN
										aTPartOnPlate[ LPP_Reject,iPlatePos].ePartStatus := PPS_Present;
									END_IF
									IF C_PROD_MODE_GOOD_PART THEN
										sProdLot.dEstimatedPartTime := TIME_TO_DWORD(TJobElapsed)  / sProdLot.dGoodQty;
										sHMIPartData.bEndOfProd := sProdLot.dGoodQty >= sProdLot.dLotQty;
									ELSE
										sProdLot.dEstimatedPartTime := TIME_TO_DWORD(TJobElapsed)  / sProdLot.dProdQty;
										sHMIPartData.bEndOfProd := sProdLot.dProdQty >= sProdLot.dLotQty;
									END_IF
									sHMIPartData.sPartStatus := sRunData.aTPartData[iHead];
									sHMIPartData.bPartReady := TRUE;
								END_IF
								CASE eDropMode OF
									LDM_DropAndGoUp:
										alrTargetPos[LA_Z1+iHead] := alrSecuredSafeZPos[iHead];
										aeMoveRobotCommand[LA_Z1+iHead] := AC_MoveAtAbsPos;
								END_CASE
								sCurrentState.eStep := SP_RunStp24;
							END_IF
						SP_RunStp24 :
							IF (sRunData.eModule = LMP_Reject OR  sRunData.eModule = LMP_Sample) AND sRejectRunData.eRejectStatus<>RS_Locked THEN
								aeMoveRobotCommand[LA_Z1+iHead] := AC_ForceStop;
							END_IF
							IF aTRobotAxis[LA_Z1+iHead].eCurrentState = AS_InPosition THEN
								IF (sRunData.eModule = LMP_Reject OR sRunData.eModule = LMP_Sample) AND eRejectRunStatus = RS_WaitRequest AND sRejectRunData.eRejectStatus=RS_Locked THEN
									eRejectRunCmd := RCR_UnlockDrawer;
								END_IF
								sOutGiveToModule.bHasGiven := TRUE;
								sCurrentState.eStep := SP_RunStp25;
							END_IF
						SP_RunStp25 :
							(* Check if right loader has taken the plate *)
							IF sInGiveToModule.bHasTaken  OR NOT bUseGiveTake THEN
								abEnableHeadVacuum[iHead] := FALSE;
								sCurrentState.eStep := SP_RunStp26;
							ELSIF sInGiveToModule.bHasNotTaken THEN
								sCurrentState.eStep := SP_RunStp28;
							END_IF
						SP_RunStp26 :
							IF aTHeadVacuum[iHead].bVacuumCorrect  THEN
								sRunData.aTPartData[iHead].bPartPresent := FALSE;
								alrTargetPos[LA_Z1+iHead] := alrSecuredSafeZPos[iHead];
								aeMoveRobotCommand[LA_Z1+iHead] := AC_MoveAtAbsPos;
								sCurrentState.eStep := SP_RunStp27;
							END_IF
						SP_RunStp27 :
							IF aTRobotAxis[LA_Z1+iHead].eCurrentState = AS_InPosition OR
									(bUse103171OptimB5MoveOnPreSafeZ AND  (aTRobotAxis[LA_Z1].lrCurrentPos < (alrSecuredSafeZPos[0]+lrPreSafeTolerance)))THEN
								(* Remove HasGiven so table can check vacuum *)
								sOutGiveToModule.bHasGiven := FALSE;
								sCurrentState.eStep := SP_RunStp1;
							END_IF
						SP_RunStp28 :
							abEnableHeadVacuum[iHead] := TRUE;
							IF aTHeadVacuum[iHead].bVacuumCorrect  THEN
								sRunData.aTPartData[iHead].bPartPresent := TRUE;
								sRunData.aTPartData[iHead].bToReject:= TRUE;
								alrTargetPos[LA_Z1+iHead] := alrSecuredSafeZPos[iHead];
								aeMoveRobotCommand[LA_Z1+iHead] := AC_MoveAtAbsPos;
								sCurrentState.eStep := SP_RunStp27;
							END_IF
						SP_RunStp30: (*Take Plate*)
							alrSecuredTarget[LA_X] := alrRobotPos[LTA_X,LTP_Lift1] +alrRobotOffset[LTA_X, LTO_Plate] + alrLiftCalibrationOffset[LTP_Lift1,LTA_X] - sPlateData.alrTakePlatePos.lrX;
							alrSecuredTarget[LA_Y] := alrRobotPos[LTA_Y,LTP_Lift1] +alrRobotOffset[LTA_Y, LTO_Plate] + alrLiftCalibrationOffset[LTP_Lift1,LTA_Y] - sPlateData.alrTakePlatePos.lrY;
							eReturnStep4SecureMove := SP_RunStp31;
							sCurrentState.eStep := SP_RunStp550;
						SP_RunStp31 :  (*Movement done*)
							IF eRobotXYTStatus = AS_InPosition THEN
								bMovePlateTakerDown := TRUE;
								sCurrentState.eStep := SP_RunStp32;
							END_IF
						SP_RunStp32 :   (*Take plate *)
							IF bPlateTakerIsDown THEN
								bEnablePlateVacuum := TRUE;
								sCurrentState.eStep := SP_RunStp33;
							END_IF
						SP_RunStp33 :
							IF TPlateVacuum.bVacuumCorrect THEN
								sRunData.bPlatePresent := TRUE;
								bMovePlateTakerDown := FALSE;
								sCurrentState.eStep := SP_RunStp34;
							END_IF
						SP_RunStp34 :
							IF bPlateTakerIsUp THEN
								sCurrentState.eStep := eReturnStep;
							END_IF
						SP_RunStp40: (*Give Plate*)
							alrRobotSpeed[LA_X] := lrSpeedWithPlate;
							alrRobotSpeed[LA_Y] := lrSpeedWithPlate;
							alrSecuredTarget[LA_X] := alrRobotPos[LTA_X,LTP_Lift2] +alrRobotOffset[LTA_X, LTO_Plate] + alrLiftCalibrationOffset[LTP_Lift2,LTA_X] - sPlateData.alrTakePlatePos.lrX - 1.5;
							alrSecuredTarget[LA_Y] := alrRobotPos[LTA_Y,LTP_Lift2] +alrRobotOffset[LTA_Y, LTO_Plate] + alrLiftCalibrationOffset[LTP_Lift2,LTA_Y] - sPlateData.alrTakePlatePos.lrY + 0;
							eReturnStep4SecureMove := SP_RunStp41;
							sCurrentState.eStep := SP_RunStp550;
						SP_RunStp41 :  (*Movement done*)
							IF eRobotXYTStatus = AS_InPosition THEN
								alrRobotSpeed := alrMaxRobotSpeed;
								bMovePlateTakerDown := TRUE;
								sCurrentState.eStep := SP_RunStp42;
							END_IF
						SP_RunStp42 :   (*Drop plate *)
							IF bPlateTakerIsDown THEN
								bEnablePlateVacuum := FALSE;
								sRunData.bPlatePresent := FALSE;
								sCurrentState.eStep := SP_RunStp43;
							END_IF
						SP_RunStp43 :
							IF TPlateVacuum.bVacuumCorrect THEN
								bMovePlateTakerDown := FALSE;
								sCurrentState.eStep := SP_RunStp44;
							END_IF
						SP_RunStp44 :
							IF bPlateTakerIsUp THEN
								sCurrentState.eStep := eReturnStep;
							END_IF
						SP_RunStp50: (*Move To Safe*)
							IF aTRobotAxis[LA_Y].lrCurrentPos <= alrYSafePosDuringRun THEN
								(* No need to move, already safe *)
								sCurrentState.eStep := SP_RunStp1;
							ELSE
								// Use secured area X
								alrSecuredTarget[LA_X] := alrUnsecuredArea[1,LA_X];
								alrSecuredTarget[LA_Y] := alrYSafePosDuringRun;
								eReturnStep4SecureMove := SP_RunStp51;
								sCurrentState.eStep := SP_RunStp550;
							END_IF
						SP_RunStp51 :  (*Movement done*)
							IF eRobotXYTStatus = AS_InPosition THEN
								sCurrentState.eStep := SP_RunStp1;
							END_IF
						SP_RunStp60: (*Cleaning*)
							IF aTRobotAxis[LA_X].lrCurrentPos <= alrRobotPos[LTA_X,LTP_CleanBrush] +alrRobotOffset[LTA_X, LTO_Z1+iHead] THEN
								alrSecuredTarget[LA_X] := alrRobotPos[LTA_X,LTP_CleanBrush] +alrRobotOffset[LTA_X, LTO_Z1+iHead] - alrCleaningOffset;
								bCleaningFromNegToPos := TRUE;
							ELSE
								alrSecuredTarget[LA_X] := alrRobotPos[LTA_X,LTP_CleanBrush] +alrRobotOffset[LTA_X, LTO_Z1+iHead] + alrCleaningOffset;
								bCleaningFromNegToPos := FALSE;
							END_IF
							alrSecuredTarget[LA_Y] := alrRobotPos[LTA_Y,LTP_CleanBrush] +alrRobotOffset[LTA_Y, LTO_Z1+iHead];
							alrTargetPos[LA_THETA] := alrRobotPos[LTA_THETA,LTP_CleanBrush] + alrRobotOffset[LTA_THETA, LTO_Z1+iHead] + lrCleaningThetaAngle;
							aeMoveRobotCommand[LA_THETA] := AC_MoveAtAbsPos;
							eReturnStep4SecureMove := SP_RunStp61;
							sCurrentState.eStep := SP_RunStp550;
						SP_RunStp61:
							IF eRobotXYTStatus = AS_InPosition THEN
								alrTargetPos[LA_Z1+iHead] := alrRobotPos[LTA_Z,LTP_CleanBrush] +alrRobotOffset[LTA_Z, LTO_Z1+iHead] - (sPartDataMMI.lrPartAndHeadHeight -  lrCalibrationPartAndHeadHeight) + sPartDataMMI.lrPartOffsetZCleaning;
								aeMoveRobotCommand[LA_Z1+iHead] := AC_MoveAtAbsPos;
								sCurrentState.eStep := SP_RunStp62;
							END_IF
						SP_RunStp62:  (*Start cleaning the part *)
							IF aTRobotAxis[LA_Z1+iHead].eCurrentState = AS_InPosition THEN
								bAspirationBrushOn := TRUE;
								alrRobotSpeed[LA_X] := lrCleaningXSpeed;
								alrRobotSpeed[LA_THETA] := lrCleaningThetaSpeed;
								IF bCleaningFromNegToPos THEN
									alrSecuredTarget[LA_X] := alrRobotPos[LTA_X,LTP_CleanBrush] +alrRobotOffset[LTA_X, LTO_Z1+iHead] + alrCleaningOffset;
								ELSE
									alrSecuredTarget[LA_X] := alrRobotPos[LTA_X,LTP_CleanBrush] +alrRobotOffset[LTA_X, LTO_Z1+iHead] - alrCleaningOffset;
								END_IF
								bCleaningThetaCw := TRUE;
								bCleaningStopTheta := FALSE;
								eReturnStep4SecureMove := SP_RunStp63;
								sCurrentState.eStep := SP_RunStp550;
							END_IF
						SP_RunStp63: (*Cleaning the part with rotation *)
							IF aTRobotAxis[LA_X].eCurrentState = AS_InPosition THEN
								IF aTRobotAxis[LA_THETA].eCurrentState = AS_InPosition THEN
									alrRobotSpeed := alrMaxRobotSpeed;
									bAspirationBrushOn := FALSE;
									sCurrentState.eStep := SP_RunStp64;
								ELSIF NOT bCleaningStopTheta THEN (* Stop theta*)
									bCleaningStopTheta := TRUE;
									aeMoveRobotCommand[LA_THETA] := AC_Stop;
								END_IF
							ELSIF aTRobotAxis[LA_THETA].eCurrentState = AS_InPosition THEN
								bCleaningThetaCw := NOT bCleaningThetaCw;
								IF bCleaningThetaCw THEN
									alrTargetPos[LA_THETA] := alrRobotPos[LTA_THETA,LTP_CleanBrush] + alrRobotOffset[LTA_THETA, LTO_Z1+iHead] + lrCleaningThetaAngle;
								ELSE
									alrTargetPos[LA_THETA] := alrRobotPos[LTA_THETA,LTP_CleanBrush] + alrRobotOffset[LTA_THETA, LTO_Z1+iHead] - lrCleaningThetaAngle;
								END_IF
								aeMoveRobotCommand[LA_THETA] := AC_MoveAtAbsPos;
							END_IF
						SP_RunStp64:
							alrTargetPos[LA_Z1+iHead] := alrSecuredSafeZPos[iHead];
							aeMoveRobotCommand[LA_Z1+iHead] := AC_MoveAtAbsPos;
							sCurrentState.eStep := SP_RunStp65;
						SP_RunStp65 :
							IF aTRobotAxis[LA_Z1+iHead].eCurrentState = AS_InPosition OR
									(bUse103171OptimB5MoveOnPreSafeZ AND  (aTRobotAxis[LA_Z1].lrCurrentPos < (alrSecuredSafeZPos[0]+lrPreSafeTolerance)))THEN
								sCurrentState.eStep := SP_RunStp1;
							END_IF
						SP_RunStp70: (* Switch plate (Lift1 must be ready for take plate ) *)
							eReturnStepSwitchPlate := eReturnStep;
							sCurrentState.eStep := SP_RunStp71;
						SP_RunStp71: (*Lift move to load pos *)
							IF eLift1RunStatus = RS_WaitRequest THEN
								CASE sLift1RunData.eLiftPos OF
									LP_OnPlateLoad:
										bDoNothing := bDoNothing;
									LP_Empty,LP_Full:
										bLift1NeedsPlate := TRUE;
										eLift1RunCmd := RCL_MoveToOpenDrawer;
									ELSE
										eLift1RunCmd := RCL_MoveToLoadPlate;
								END_CASE
							END_IF
							IF eLift2RunStatus = RS_WaitRequest THEN
								CASE sLift2RunData.eLiftPos OF
									LP_OnPlateLoad:
										bDoNothing := bDoNothing;
									LP_Full:
										bLift2NeedsPlate := TRUE;
										eLift2RunCmd := RCL_MoveToOpenDrawer;
									ELSE
										eLift2RunCmd := RCL_MoveToLoadPlate;
								END_CASE
							END_IF
							IF eLift1RunStatus = RS_WaitRequest AND sLift1RunData.eLiftPos = LP_OnPlateLoad AND
								eLift2RunStatus = RS_WaitRequest AND sLift2RunData.eLiftPos = LP_OnPlateLoad THEN
								sCurrentState.eStep := SP_RunStp72;
							END_IF
						SP_RunStp72:
							IF NOT sRunData.bPlatePresent THEN
								//abCopySwitchFromPlate := TRUE;
								abResetPlateState[LPP_Lift1] := TRUE;
								sCurrentState.eStep := SP_RunStp30; (* Call Take plate *)
								eReturnStep := SP_RunStp72;
							ELSE
								sCurrentState.eStep := SP_RunStp73;
							END_IF
						SP_RunStp73:
							abResetPlateState[LPP_Lift2] := TRUE;
							sCurrentState.eStep := SP_RunStp40; (* Call Give plate *)
							eReturnStep := SP_RunStp74;
						SP_RunStp74:
							FOR i := 0 TO sPlateData.iNbPartOnPlate-1 DO
								aTPartOnPlate[LPP_Lift2,i].ePartStatus := PPS_Absent;
							END_FOR
							//abCopySwitchToPlate := TRUE;
							iPlatePos := 0;
							eLift1RunCmd := RCL_MoveToPlate;
							eLift2RunCmd := RCL_MoveToPlate;
							sCurrentState.eStep := SP_RunStp75;
						SP_RunStp75: (*Lift move to plate pos *)
							IF eLift1RunStatus = RS_WaitRequest AND eLift2RunStatus = RS_WaitRequest THEN
								sCurrentState.eStep := eReturnStepSwitchPlate;
							END_IF
						SP_RunStp100 : (*Prepare for take part*)
						testLD := sRunData.eModule;
							CASE sRunData.eModule OF
								LMP_Lift1:
									sCurrentState.eStep := SP_RunStp101;
								LMP_Table:
									sCurrentState.eStep := SP_RunStp170;
								LMP_TurnOverFix:
									sCurrentState.eStep := SP_RunStp180;
							END_CASE
						SP_RunStp101: (* Check Lift Status*)
							IF eLift1RunStatus = RS_WaitRequest THEN
								CASE sLift1RunData.eLiftPos OF
									LP_OnPlate:
										iPlatePos := 0;
										sCurrentState.eStep := SP_RunStp102;
									LP_Full,LP_Empty:
										bLift1NeedsPlate := TRUE;
										eLift1RunCmd := RCL_MoveToOpenDrawer;
									ELSE
										eLift1RunCmd := RCL_MoveToPlate;
								END_CASE
							END_IF
						SP_RunStp102: (*Check part status*)
							bFoundPlatePos := FALSE;
							WHILE (iPlatePos < sPlateData.iNbPartOnPlate) DO
								IF aTPartOnPlate[LPP_Lift1,iPlatePos].ePartStatus = PPS_Present OR aTPartOnPlate[LPP_Lift1,iPlatePos].ePartStatus = PPS_Undefined THEN
									bFoundPlatePos := TRUE;
									EXIT;
								ELSE
									iPlatePos := iPlatePos + 1;
								END_IF
							END_WHILE
							IF NOT bFoundPlatePos THEN
								(* Goto switch plate *)
								sCurrentState.eStep := SP_RunStp150;
							ELSE
								IF bDisableVision THEN
									aTPartOnPlate[LPP_Lift1,iPlatePos].ePartStatus := PPS_Present;
									sCurrentState.eStep := SP_RunStp110;
								ELSE
									bRetryVision := TRUE;
									iScanTry := 0;
									sCurrentState.eStep := SP_RunStp103;
								END_IF
							END_IF
						SP_RunStp103: (*Scan Vision Part Position *)
							alrSecuredTarget[LA_X] := alrRobotPos[LTA_X,LTP_Lift1] + alrRobotOffset[LTA_X, LTO_Vision] + alrLiftCalibrationOffset[LTP_Lift1,LTA_X]  - sPlateData.alrPartOnPlate[iPlatePos].lrX ;
							alrSecuredTarget[LA_Y] := alrRobotPos[LTA_Y,LTP_Lift1] + alrRobotOffset[LTA_Y, LTO_Vision] + alrLiftCalibrationOffset[LTP_Lift1,LTA_Y] - sPlateData.alrPartOnPlate[iPlatePos].lrY ;
							TVisionWaitStab(IN := FALSE);
							iVisionScanModel := 0;
							eReturnStep4SecureMove := SP_RunStp104;
							sCurrentState.eStep := SP_RunStp550;
						SP_RunStp104:
							IF eRobotXYTStatus = AS_InPosition THEN
								TVisionWaitStab(IN := TRUE, PT := TVisionWaitStabTime);
								IF TVisionWaitStab.Q THEN
									eVisionRunCmd := RCV_GrabImage;
									sCurrentState.eStep := SP_RunStp105;
								END_IF
							END_IF
						SP_RunStp105: (* Move to pre-take position *)
							IF eVisionRunStatus = RS_WaitRequest THEN
								IF bUse103171OptimB5PreMoveXY THEN
									alrSecuredTarget[LA_X] := alrRobotPos[LTA_X,LTP_Lift1] + alrRobotOffset[LTA_X, iHead] + alrLiftCalibrationOffset[LTP_Lift1,LTA_X]  -  sPlateData.alrPartOnPlate[iPlatePos].lrX;
									alrSecuredTarget[LA_Y] := alrRobotPos[LTA_Y,LTP_Lift1] + alrRobotOffset[LTA_Y, iHead] + alrLiftCalibrationOffset[LTP_Lift1,LTA_Y] - sPlateData.alrPartOnPlate[iPlatePos].lrY;
									alrTargetPos[LA_THETA] := alrRobotPos[LTA_THETA,LTP_TableSideALayering1] + alrRobotOffset[LTA_THETA, iHead];
									aeMoveRobotCommand[LA_THETA] := AC_MoveAtAbsPos;
								END_IF
								sRunDataVision.iUseModel := aiVisionModelPart[iVisionScanModel];
								eVisionRunCmd := RCV_AnalyseImage;
								eReturnStep4SecureMove := SP_RunStp109;
								sCurrentState.eStep := SP_RunStp550;
							END_IF
						SP_RunStp109: (* Check for part *)
							IF eVisionRunStatus = RS_WaitRequest THEN
								IF sRunDataVision.TVisionPartData.bPresent AND sRunDataVision.TVisionPartData.bValid THEN
									(* Found valide part *)
									bBadPartDetected := FALSE;
									aTPartOnPlate[LPP_Lift1,iPlatePos].ePartStatus := PPS_Present;
									sCurrentState.eStep := SP_RunStp110;
								ELSIF sRunDataVision.TVisionPartData.bPresent AND NOT sRunDataVision.TVisionPartData.bValid THEN
									(* Found bad part *)
									IF iScanTry < iScanTryMax THEN
										iScanTry := iScanTry + 1;
										bBadPartDetected := FALSE;
										sCurrentState.eStep := SP_RunStp103;
									ELSE
										aTPartOnPlate[LPP_Lift1,iPlatePos].ePartStatus := PPS_BadPart;
										//iPlatePos := iPlatePos + 1;
										//sCurrentState.eStep := SP_RunStp102;
										bBadPartDetected := TRUE;
										sCurrentState.eStep := SP_RunStp110;
									END_IF
									
								ELSE
									(* No part *)
									aTPartOnPlate[LPP_Lift1,iPlatePos].ePartStatus := PPS_Absent;
									iPlatePos := iPlatePos + 1;
									sCurrentState.eStep := SP_RunStp102;

